LIN {X -0.019,Y -142.969,Z 1935.171,A 0.000,B 0.000,C 90.000,E1 210.846} C_DIS
LIN {X 0.034,Y -141.596,Z 1935.151,A 0.000,B 0.000,C 90.000,E1 207.129} C_DIS
LIN {X -0.051,Y -139.421,Z 1935.115,A 0.000,B 0.000,C 90.000,E1 200.663} C_DIS
LIN {X 0.000,Y -139.148,Z 1935.104,A 0.000,B 0.000,C 90.000,E1 198.779} C_DIS
LIN {X 0.022,Y -138.345,Z 1935.058,A 0.000,B 0.000,C 90.000,E1 190.366} C_DIS
LIN {X 0.008,Y -139.487,Z 1935.006,A 0.000,B 0.000,C 90.000,E1 181.031} C_DIS
LIN {X -0.052,Y -141.088,Z 1934.975,A 0.000,B 0.000,C 90.000,E1 175.469} C_DIS
LIN {X 0.043,Y -142.466,Z 1934.959,A 0.000,B 0.000,C 90.000,E1 172.648} C_DIS
LIN {X -0.009,Y -144.710,Z 1934.934,A 0.000,B 0.000,C 90.000,E1 168.049} C_DIS
LIN {X -0.058,Y -147.309,Z 1934.913,A 0.000,B 0.000,C 90.000,E1 164.393} C_DIS
LIN {X -0.043,Y -150.630,Z 1934.888,A 0.000,B 0.000,C 90.000,E1 159.826} C_DIS
LIN {X 0.033,Y -154.106,Z 1934.868,A 0.000,B 0.000,C 90.000,E1 156.177} C_DIS
LIN {X -0.042,Y -157.530,Z 1934.848,A 0.000,B 0.000,C 90.000,E1 152.615} C_DIS
LIN {X -0.099,Y -161.765,Z 1934.828,A 0.000,B 0.000,C 90.000,E1 149.076} C_DIS
LIN {X 0.007,Y -165.958,Z 1934.808,A 0.000,B 0.000,C 90.000,E1 145.515} C_DIS
LIN {X 0.003,Y -170.951,Z 1934.789,A 0.000,B 0.000,C 90.000,E1 142.029} C_DIS
LIN {X 0.055,Y -175.820,Z 1934.770,A 0.000,B 0.000,C 90.000,E1 138.566} C_DIS
LIN {X 0.051,Y -181.426,Z 1934.751,A 0.000,B 0.000,C 90.000,E1 135.162} C_DIS
LIN {X -0.075,Y -186.930,Z 1934.732,A 0.000,B 0.000,C 90.000,E1 131.838} C_DIS
LIN {X -0.003,Y -191.509,Z 1934.719,A 0.000,B 0.000,C 90.000,E1 129.322} C_DIS
LIN {X 0.082,Y -197.374,Z 1934.700,A 0.000,B 0.000,C 90.000,E1 126.011} C_DIS
LIN {X 0.007,Y -200.649,Z 1934.691,A 0.000,B 0.000,C 90.000,E1 124.405} C_DIS
LIN {X -0.083,Y -206.533,Z 1934.673,A 0.000,B 0.000,C 90.000,E1 121.209} C_DIS
LIN {X 0.011,Y -209.824,Z 1934.664,A 0.000,B 0.000,C 90.000,E1 119.589} C_DIS
LIN {X -0.063,Y -217.182,Z 1934.642,A 0.000,B 0.000,C 90.000,E1 115.668} C_DIS
LIN {X -0.110,Y -218.809,Z 1934.638,A 0.000,B 0.000,C 90.000,E1 114.899} C_DIS
LIN {X 0.031,Y -224.195,Z 1934.621,A 0.000,B 0.000,C 90.000,E1 111.791} C_DIS
LIN {X 0.113,Y -284.154,Z 1934.621,A 0.000,B 0.000,C 90.000,E1 111.770} C_DIS
LIN {X 0.017,Y -285.333,Z 1934.621,A 0.000,B 0.000,C 90.000,E1 111.770} C_DIS
LIN {X -0.012,Y -288.714,Z 1934.620,A 0.000,B 0.000,C 90.000,E1 111.642} C_DIS
LIN {X -0.078,Y -291.984,Z 1934.619,A 0.000,B 0.000,C 90.000,E1 111.408} C_DIS
LIN {X 0.114,Y -295.661,Z 1934.616,A 0.000,B 0.000,C 90.000,E1 110.918} C_DIS
LIN {X -0.073,Y -310.921,Z 1934.602,A 0.000,B 0.000,C 90.000,E1 108.308} C_DIS
LIN {X 0.068,Y -325.651,Z 1934.589,A 0.000,B 0.000,C 90.000,E1 106.024} C_DIS
LIN {X 0.158,Y -339.472,Z 1934.579,A 0.000,B 0.000,C 90.000,E1 104.120} C_DIS
LIN {X 0.015,Y -354.484,Z 1934.568,A 0.000,B 0.000,C 90.000,E1 102.299} C_DIS
LIN {X 0.159,Y -372.954,Z 1934.557,A 0.000,B 0.000,C 90.000,E1 100.254} C_DIS
LIN {X -0.077,Y -391.821,Z 1934.547,A 0.000,B 0.000,C 90.000,E1 98.454} C_DIS
LIN {X -0.060,Y -411.099,Z 1934.538,A 0.000,B 0.000,C 90.000,E1 96.777} C_DIS
LIN {X -0.118,Y -433.506,Z 1934.528,A 0.000,B 0.000,C 90.000,E1 95.049} C_DIS
LIN {X -0.139,Y -439.166,Z 1934.526,A 0.000,B 0.000,C 90.000,E1 94.645} C_DIS
LIN {X -0.149,Y -443.334,Z 1934.523,A 0.000,B 0.000,C 90.000,E1 94.245} C_DIS
LIN {X 0.181,Y -445.054,Z 1934.522,A 0.000,B 0.000,C 90.000,E1 93.955} C_DIS
LIN {X 0.036,Y -446.375,Z 1934.521,A 0.000,B 0.000,C 90.000,E1 93.726} C_DIS
LIN {X -0.039,Y -448.200,Z 1934.518,A 0.000,B 0.000,C 90.000,E1 93.212} C_DIS
LIN {X -0.081,Y -448.963,Z 1934.515,A 0.000,B 0.000,C 90.000,E1 92.694} C_DIS
LIN {X -0.135,Y -448.790,Z 1934.512,A 0.000,B 0.000,C 90.000,E1 92.178} C_DIS
LIN {X -0.168,Y -447.662,Z 1934.509,A 0.000,B 0.000,C 90.000,E1 91.661} C_DIS
LIN {X 0.032,Y -446.690,Z 1934.508,A 0.000,B 0.000,C 90.000,E1 91.375} C_DIS
LIN {X -0.216,Y -445.387,Z 1934.506,A 0.000,B 0.000,C 90.000,E1 91.146} C_DIS
LIN {X 0.160,Y -433.910,Z 1934.496,A 0.000,B 0.000,C 90.000,E1 89.255} C_DIS
LIN {X 0.177,Y -423.887,Z 1934.487,A 0.000,B 0.000,C 90.000,E1 87.650} C_DIS
LIN {X 0.137,Y -412.109,Z 1934.477,A 0.000,B 0.000,C 90.000,E1 85.755} C_DIS
LIN {X -0.196,Y -401.950,Z 1934.467,A 0.000,B 0.000,C 90.000,E1 84.147} C_DIS
LIN {X -0.211,Y -389.964,Z 1934.456,A 0.000,B 0.000,C 90.000,E1 82.186} C_DIS
LIN {X 0.022,Y -378.082,Z 1934.445,A 0.000,B 0.000,C 90.000,E1 80.151} C_DIS
LIN {X 0.037,Y -363.093,Z 1934.431,A 0.000,B 0.000,C 90.000,E1 77.521} C_DIS
LIN {X 0.108,Y -345.897,Z 1934.412,A 0.000,B 0.000,C 90.000,E1 74.212} C_DIS
LIN {X 0.052,Y -333.963,Z 1934.399,A 0.000,B 0.000,C 90.000,E1 71.764} C_DIS
LIN {X 0.061,Y -323.718,Z 1934.387,A 0.000,B 0.000,C 90.000,E1 69.571} C_DIS
LIN {X 0.153,Y -309.663,Z 1934.369,A 0.000,B 0.000,C 90.000,E1 66.357} C_DIS
LIN {X 0.003,Y -300.191,Z 1934.356,A 0.000,B 0.000,C 90.000,E1 64.101} C_DIS
LIN {X -0.115,Y -288.155,Z 1934.339,A 0.000,B 0.000,C 90.000,E1 61.129} C_DIS
LIN {X -0.015,Y -280.090,Z 1934.328,A 0.000,B 0.000,C 90.000,E1 59.076} C_DIS
LIN {X 0.158,Y -270.556,Z 1934.315,A 0.000,B 0.000,C 90.000,E1 56.628} C_DIS
LIN {X 0.074,Y -263.707,Z 1934.305,A 0.000,B 0.000,C 90.000,E1 54.895} C_DIS
LIN {X -0.006,Y -252.710,Z 1934.289,A 0.000,B 0.000,C 90.000,E1 52.065} C_DIS
LIN {X -0.086,Y -243.127,Z 1934.275,A 0.000,B 0.000,C 90.000,E1 49.542} C_DIS
LIN {X 0.066,Y -232.480,Z 1934.259,A 0.000,B 0.000,C 90.000,E1 46.539} C_DIS
LIN {X -0.064,Y -222.206,Z 1934.242,A 0.000,B 0.000,C 90.000,E1 43.542} C_DIS
LIN {X 0.099,Y -211.300,Z 1934.222,A 0.000,B 0.000,C 90.000,E1 40.011} C_DIS
LIN {X -0.042,Y -203.498,Z 1934.207,A 0.000,B 0.000,C 90.000,E1 37.282} C_DIS
LIN {X -0.047,Y -195.382,Z 1934.189,A 0.000,B 0.000,C 90.000,E1 34.072} C_DIS
LIN {X -0.029,Y -188.013,Z 1934.171,A 0.000,B 0.000,C 90.000,E1 30.797} C_DIS
LIN {X 0.006,Y -181.382,Z 1934.153,A 0.000,B 0.000,C 90.000,E1 27.462} C_DIS
LIN {X -0.041,Y -176.866,Z 1934.139,A 0.000,B 0.000,C 90.000,E1 24.951} C_DIS
LIN {X -0.019,Y -171.587,Z 1934.120,A 0.000,B 0.000,C 90.000,E1 21.535} C_DIS
LIN {X 0.071,Y -167.096,Z 1934.100,A 0.000,B 0.000,C 90.000,E1 18.055} C_DIS
LIN {X 0.002,Y -163.458,Z 1934.081,A 0.000,B 0.000,C 90.000,E1 14.592} C_DIS
LIN {X -0.011,Y -159.746,Z 1934.057,A 0.000,B 0.000,C 90.000,E1 10.197} C_DIS
LIN {X 0.050,Y -157.186,Z 1934.032,A 0.000,B 0.000,C 90.000,E1 5.739} C_DIS
LIN {X -0.028,Y -154.901,Z 1933.997,A 0.000,B 0.000,C 90.000,E1 359.542} C_DIS
LIN {X 0.057,Y -154.146,Z 1933.953,A 0.000,B 0.000,C 90.000,E1 351.432} C_DIS
LIN {X -0.021,Y -155.869,Z 1933.913,A 0.000,B 0.000,C 90.000,E1 344.283} C_DIS
LIN {X 0.041,Y -158.583,Z 1933.883,A 0.000,B 0.000,C 90.000,E1 338.901} C_DIS
LIN {X 0.055,Y -162.176,Z 1933.858,A 0.000,B 0.000,C 90.000,E1 334.460} C_DIS
LIN {X -0.038,Y -166.049,Z 1933.839,A 0.000,B 0.000,C 90.000,E1 330.973} C_DIS
LIN {X 0.060,Y -170.918,Z 1933.819,A 0.000,B 0.000,C 90.000,E1 327.454} C_DIS
LIN {X -0.028,Y -175.211,Z 1933.805,A 0.000,B 0.000,C 90.000,E1 324.895} C_DIS
LIN {X 0.023,Y -180.173,Z 1933.791,A 0.000,B 0.000,C 90.000,E1 322.316} C_DIS
LIN {X 0.022,Y -186.029,Z 1933.777,A 0.000,B 0.000,C 90.000,E1 319.784} C_DIS
LIN {X -0.012,Y -191.640,Z 1933.765,A 0.000,B 0.000,C 90.000,E1 317.715} C_DIS
LIN {X 0.024,Y -199.313,Z 1933.751,A 0.000,B 0.000,C 90.000,E1 315.243} C_DIS
LIN {X -0.075,Y -207.901,Z 1933.738,A 0.000,B 0.000,C 90.000,E1 312.852} C_DIS
LIN {X -0.095,Y -218.960,Z 1933.723,A 0.000,B 0.000,C 90.000,E1 310.092} C_DIS
LIN {X -0.031,Y -232.882,Z 1933.705,A 0.000,B 0.000,C 90.000,E1 306.996} C_DIS
LIN {X 0.030,Y -247.942,Z 1933.689,A 0.000,B 0.000,C 90.000,E1 303.992} C_DIS
LIN {X 0.080,Y -259.865,Z 1933.677,A 0.000,B 0.000,C 90.000,E1 301.799} C_DIS
LIN {X 0.084,Y -271.928,Z 1933.665,A 0.000,B 0.000,C 90.000,E1 299.667} C_DIS
LIN {X -0.143,Y -281.824,Z 1933.655,A 0.000,B 0.000,C 90.000,E1 297.975} C_DIS
LIN {X 0.029,Y -291.425,Z 1933.646,A 0.000,B 0.000,C 90.000,E1 296.232} C_DIS
LIN {X 0.109,Y -296.837,Z 1933.640,A 0.000,B 0.000,C 90.000,E1 295.207} C_DIS
LIN {X 0.110,Y -301.639,Z 1933.635,A 0.000,B 0.000,C 90.000,E1 294.207} C_DIS
LIN {X -0.004,Y -304.447,Z 1933.631,A 0.000,B 0.000,C 90.000,E1 293.567} C_DIS
LIN {X 0.057,Y -306.850,Z 1933.627,A 0.000,B 0.000,C 90.000,E1 292.898} C_DIS
LIN {X -0.030,Y -308.861,Z 1933.624,A 0.000,B 0.000,C 90.000,E1 292.259} C_DIS
LIN {X 0.058,Y -310.530,Z 1933.620,A 0.000,B 0.000,C 90.000,E1 291.589} C_DIS
LIN {X -0.129,Y -311.874,Z 1933.616,A 0.000,B 0.000,C 90.000,E1 290.972} C_DIS
LIN {X -0.014,Y -312.871,Z 1933.613,A 0.000,B 0.000,C 90.000,E1 290.301} C_DIS
LIN {X 0.111,Y -313.512,Z 1933.609,A 0.000,B 0.000,C 90.000,E1 289.631} C_DIS
LIN {X -0.158,Y -313.857,Z 1933.606,A 0.000,B 0.000,C 90.000,E1 289.033} C_DIS
LIN {X -0.023,Y -313.847,Z 1933.602,A 0.000,B 0.000,C 90.000,E1 288.362} C_DIS
LIN {X 0.111,Y -313.460,Z 1933.598,A 0.000,B 0.000,C 90.000,E1 287.692} C_DIS
LIN {X 0.150,Y -312.644,Z 1933.595,A 0.000,B 0.000,C 90.000,E1 287.040} C_DIS
LIN {X -0.110,Y -311.343,Z 1933.591,A 0.000,B 0.000,C 90.000,E1 286.441} C_DIS
LIN {X -0.075,Y -309.501,Z 1933.588,A 0.000,B 0.000,C 90.000,E1 285.788} C_DIS
LIN {X -0.048,Y -307.046,Z 1933.584,A 0.000,B 0.000,C 90.000,E1 285.134} C_DIS
LIN {X -0.039,Y -303.810,Z 1933.580,A 0.000,B 0.000,C 90.000,E1 284.481} C_DIS
LIN {X -0.081,Y -296.077,Z 1933.573,A 0.000,B 0.000,C 90.000,E1 283.175} C_DIS
LIN {X 0.005,Y -290.833,Z 1933.568,A 0.000,B 0.000,C 90.000,E1 282.187} C_DIS
LIN {X -0.087,Y -286.473,Z 1933.564,A 0.000,B 0.000,C 90.000,E1 281.535} C_DIS
LIN {X 0.018,Y -281.136,Z 1933.560,A 0.000,B 0.000,C 90.000,E1 280.838} C_DIS
LIN {X 0.016,Y -274.907,Z 1933.557,A 0.000,B 0.000,C 90.000,E1 280.197} C_DIS
LIN {X 0.068,Y -268.464,Z 1933.553,A 0.000,B 0.000,C 90.000,E1 279.613} C_DIS
LIN {X -0.143,Y -261.822,Z 1933.551,A 0.000,B 0.000,C 90.000,E1 279.151} C_DIS
LIN {X -0.032,Y -255.092,Z 1933.548,A 0.000,B 0.000,C 90.000,E1 278.681} C_DIS
LIN {X 0.029,Y -248.149,Z 1933.546,A 0.000,B 0.000,C 90.000,E1 278.276} C_DIS
LIN {X 0.084,Y -240.671,Z 1933.544,A 0.000,B 0.000,C 90.000,E1 277.936} C_DIS
LIN {X -0.018,Y -232.620,Z 1933.543,A 0.000,B 0.000,C 90.000,E1 277.701} C_DIS
LIN {X -0.096,Y -221.950,Z 1933.542,A 0.000,B 0.000,C 90.000,E1 277.530} C_DIS
LIN {X -0.033,Y -216.160,Z 1933.541,A 0.000,B 0.000,C 90.000,E1 277.466} C_DIS
LIN {X -0.058,Y -180.199,Z 1933.541,A 0.000,B 0.000,C 90.000,E1 277.466} C_DIS
LIN {X 0.058,Y -181.027,Z 1933.530,A 0.000,B 0.000,C 90.000,E1 275.391} C_DIS
LIN {X 0.033,Y -181.578,Z 1933.502,A 0.000,B 0.000,C 90.000,E1 270.344} C_DIS
LIN {X 0.009,Y -180.904,Z 1933.474,A 0.000,B 0.000,C 90.000,E1 265.298} C_DIS
LIN {X -0.042,Y -180.245,Z 1933.464,A 0.000,B 0.000,C 90.000,E1 263.628} C_DIS
LIN {X -0.023,Y -178.732,Z 1933.441,A 0.000,B 0.000,C 90.000,E1 259.398} C_DIS
LIN {X 0.045,Y -175.780,Z 1933.413,A 0.000,B 0.000,C 90.000,E1 254.283} C_DIS
LIN {X 0.032,Y -171.964,Z 1933.384,A 0.000,B 0.000,C 90.000,E1 249.156} C_DIS
LIN {X 0.069,Y -171.361,Z 1933.380,A 0.000,B 0.000,C 90.000,E1 248.284} C_DIS
LIN {X 0.046,Y -167.610,Z 1933.355,A 0.000,B 0.000,C 90.000,E1 243.973} C_DIS
LIN {X 0.059,Y -166.257,Z 1933.346,A 0.000,B 0.000,C 90.000,E1 242.231} C_DIS
LIN {X 0.046,Y -163.011,Z 1933.326,A 0.000,B 0.000,C 90.000,E1 238.742} C_DIS
LIN {X -0.040,Y -160.934,Z 1933.312,A 0.000,B 0.000,C 90.000,E1 236.135} C_DIS
LIN {X 0.069,Y -157.694,Z 1933.292,A 0.000,B 0.000,C 90.000,E1 232.557} C_DIS
LIN {X 0.008,Y -155.733,Z 1933.277,A 0.000,B 0.000,C 90.000,E1 229.908} C_DIS
LIN {X 0.061,Y -151.992,Z 1933.252,A 0.000,B 0.000,C 90.000,E1 225.405} C_DIS
LIN {X 0.077,Y -150.237,Z 1933.237,A 0.000,B 0.000,C 90.000,E1 222.690} C_DIS
LIN {X -0.001,Y -146.997,Z 1933.212,A 0.000,B 0.000,C 90.000,E1 218.177} C_DIS
LIN {X -0.010,Y -145.582,Z 1933.197,A 0.000,B 0.000,C 90.000,E1 215.438} C_DIS
LIN {X -0.016,Y -142.970,Z 1933.171,A 0.000,B 0.000,C 90.000,E1 210.846} C_DIS
LIN {X 0.037,Y -141.597,Z 1933.151,A 0.000,B 0.000,C 90.000,E1 207.129} C_DIS
LIN {X -0.046,Y -139.422,Z 1933.115,A 0.000,B 0.000,C 90.000,E1 200.663} C_DIS
LIN {X 0.004,Y -139.150,Z 1933.104,A 0.000,B 0.000,C 90.000,E1 198.779} C_DIS
LIN {X 0.026,Y -138.346,Z 1933.058,A 0.000,B 0.000,C 90.000,E1 190.366} C_DIS
LIN {X 0.012,Y -139.487,Z 1933.006,A 0.000,B 0.000,C 90.000,E1 181.031} C_DIS
LIN {X -0.048,Y -141.088,Z 1932.975,A 0.000,B 0.000,C 90.000,E1 175.469} C_DIS
LIN {X 0.047,Y -142.464,Z 1932.959,A 0.000,B 0.000,C 90.000,E1 172.648} C_DIS
LIN {X -0.005,Y -144.709,Z 1932.934,A 0.000,B 0.000,C 90.000,E1 168.049} C_DIS
LIN {X -0.054,Y -147.308,Z 1932.913,A 0.000,B 0.000,C 90.000,E1 164.393} C_DIS
LIN {X -0.039,Y -150.628,Z 1932.888,A 0.000,B 0.000,C 90.000,E1 159.826} C_DIS
LIN {X 0.037,Y -154.105,Z 1932.868,A 0.000,B 0.000,C 90.000,E1 156.177} C_DIS
LIN {X -0.039,Y -157.528,Z 1932.848,A 0.000,B 0.000,C 90.000,E1 152.615} C_DIS
LIN {X -0.095,Y -161.763,Z 1932.828,A 0.000,B 0.000,C 90.000,E1 149.076} C_DIS
LIN {X 0.011,Y -165.957,Z 1932.808,A 0.000,B 0.000,C 90.000,E1 145.515} C_DIS
LIN {X 0.008,Y -170.948,Z 1932.789,A 0.000,B 0.000,C 90.000,E1 142.029} C_DIS
LIN {X 0.059,Y -175.817,Z 1932.770,A 0.000,B 0.000,C 90.000,E1 138.566} C_DIS
LIN {X 0.055,Y -181.424,Z 1932.751,A 0.000,B 0.000,C 90.000,E1 135.162} C_DIS
LIN {X -0.071,Y -186.929,Z 1932.732,A 0.000,B 0.000,C 90.000,E1 131.838} C_DIS
LIN {X 0.002,Y -191.506,Z 1932.719,A 0.000,B 0.000,C 90.000,E1 129.322} C_DIS
LIN {X 0.087,Y -197.371,Z 1932.700,A 0.000,B 0.000,C 90.000,E1 126.011} C_DIS
LIN {X 0.011,Y -200.647,Z 1932.691,A 0.000,B 0.000,C 90.000,E1 124.405} C_DIS
LIN {X -0.079,Y -206.530,Z 1932.673,A 0.000,B 0.000,C 90.000,E1 121.209} C_DIS
LIN {X 0.015,Y -209.822,Z 1932.664,A 0.000,B 0.000,C 90.000,E1 119.589} C_DIS
LIN {X -0.059,Y -217.180,Z 1932.642,A 0.000,B 0.000,C 90.000,E1 115.668} C_DIS
LIN {X -0.105,Y -218.806,Z 1932.638,A 0.000,B 0.000,C 90.000,E1 114.899} C_DIS
LIN {X 0.036,Y -224.194,Z 1932.621,A 0.000,B 0.000,C 90.000,E1 111.791} C_DIS
LIN {X 0.119,Y -284.134,Z 1932.621,A 0.000,B 0.000,C 90.000,E1 111.770} C_DIS
LIN {X 0.022,Y -285.319,Z 1932.621,A 0.000,B 0.000,C 90.000,E1 111.770} C_DIS
LIN {X -0.003,Y -288.698,Z 1932.620,A 0.000,B 0.000,C 90.000,E1 111.642} C_DIS
LIN {X -0.068,Y -291.966,Z 1932.619,A 0.000,B 0.000,C 90.000,E1 111.408} C_DIS
LIN {X 0.128,Y -295.643,Z 1932.616,A 0.000,B 0.000,C 90.000,E1 110.918} C_DIS
LIN {X -0.056,Y -310.901,Z 1932.602,A 0.000,B 0.000,C 90.000,E1 108.308} C_DIS
LIN {X 0.087,Y -325.627,Z 1932.589,A 0.000,B 0.000,C 90.000,E1 106.024} C_DIS
LIN {X 0.176,Y -339.447,Z 1932.579,A 0.000,B 0.000,C 90.000,E1 104.120} C_DIS
LIN {X 0.035,Y -354.456,Z 1932.568,A 0.000,B 0.000,C 90.000,E1 102.299} C_DIS
LIN {X 0.176,Y -372.924,Z 1932.557,A 0.000,B 0.000,C 90.000,E1 100.254} C_DIS
LIN {X -0.060,Y -391.792,Z 1932.547,A 0.000,B 0.000,C 90.000,E1 98.454} C_DIS
LIN {X -0.043,Y -411.070,Z 1932.538,A 0.000,B 0.000,C 90.000,E1 96.777} C_DIS
LIN {X -0.102,Y -433.476,Z 1932.528,A 0.000,B 0.000,C 90.000,E1 95.049} C_DIS
LIN {X -0.123,Y -439.135,Z 1932.526,A 0.000,B 0.000,C 90.000,E1 94.645} C_DIS
LIN {X -0.134,Y -443.311,Z 1932.523,A 0.000,B 0.000,C 90.000,E1 94.245} C_DIS
LIN {X 0.198,Y -445.032,Z 1932.522,A 0.000,B 0.000,C 90.000,E1 93.955} C_DIS
LIN {X 0.055,Y -446.353,Z 1932.521,A 0.000,B 0.000,C 90.000,E1 93.726} C_DIS
LIN {X -0.020,Y -448.182,Z 1932.518,A 0.000,B 0.000,C 90.000,E1 93.212} C_DIS
LIN {X -0.062,Y -448.948,Z 1932.515,A 0.000,B 0.000,C 90.000,E1 92.694} C_DIS
LIN {X -0.116,Y -448.778,Z 1932.512,A 0.000,B 0.000,C 90.000,E1 92.178} C_DIS
LIN {X -0.149,Y -447.653,Z 1932.509,A 0.000,B 0.000,C 90.000,E1 91.661} C_DIS
LIN {X 0.050,Y -446.682,Z 1932.508,A 0.000,B 0.000,C 90.000,E1 91.375} C_DIS
LIN {X -0.197,Y -445.381,Z 1932.506,A 0.000,B 0.000,C 90.000,E1 91.146} C_DIS
LIN {X 0.178,Y -433.905,Z 1932.496,A 0.000,B 0.000,C 90.000,E1 89.255} C_DIS
LIN {X 0.194,Y -423.883,Z 1932.487,A 0.000,B 0.000,C 90.000,E1 87.650} C_DIS
LIN {X 0.154,Y -412.105,Z 1932.477,A 0.000,B 0.000,C 90.000,E1 85.755} C_DIS
LIN {X -0.180,Y -401.947,Z 1932.467,A 0.000,B 0.000,C 90.000,E1 84.147} C_DIS
LIN {X -0.195,Y -389.961,Z 1932.456,A 0.000,B 0.000,C 90.000,E1 82.186} C_DIS
LIN {X 0.037,Y -378.076,Z 1932.445,A 0.000,B 0.000,C 90.000,E1 80.151} C_DIS
LIN {X 0.052,Y -363.086,Z 1932.431,A 0.000,B 0.000,C 90.000,E1 77.521} C_DIS
LIN {X 0.122,Y -345.888,Z 1932.412,A 0.000,B 0.000,C 90.000,E1 74.212} C_DIS
LIN {X 0.065,Y -333.955,Z 1932.399,A 0.000,B 0.000,C 90.000,E1 71.764} C_DIS
LIN {X 0.074,Y -323.708,Z 1932.387,A 0.000,B 0.000,C 90.000,E1 69.571} C_DIS
LIN {X 0.165,Y -309.651,Z 1932.369,A 0.000,B 0.000,C 90.000,E1 66.357} C_DIS
LIN {X 0.015,Y -300.178,Z 1932.356,A 0.000,B 0.000,C 90.000,E1 64.101} C_DIS
LIN {X -0.105,Y -288.140,Z 1932.339,A 0.000,B 0.000,C 90.000,E1 61.129} C_DIS
LIN {X -0.005,Y -280.075,Z 1932.328,A 0.000,B 0.000,C 90.000,E1 59.076} C_DIS
LIN {X 0.167,Y -270.544,Z 1932.315,A 0.000,B 0.000,C 90.000,E1 56.628} C_DIS
LIN {X 0.082,Y -263.695,Z 1932.305,A 0.000,B 0.000,C 90.000,E1 54.895} C_DIS
LIN {X 0.002,Y -252.701,Z 1932.289,A 0.000,B 0.000,C 90.000,E1 52.065} C_DIS
LIN {X -0.079,Y -243.117,Z 1932.275,A 0.000,B 0.000,C 90.000,E1 49.542} C_DIS
LIN {X 0.072,Y -232.468,Z 1932.259,A 0.000,B 0.000,C 90.000,E1 46.539} C_DIS
LIN {X -0.058,Y -222.193,Z 1932.242,A 0.000,B 0.000,C 90.000,E1 43.542} C_DIS
LIN {X 0.104,Y -211.288,Z 1932.222,A 0.000,B 0.000,C 90.000,E1 40.011} C_DIS
LIN {X -0.037,Y -203.488,Z 1932.207,A 0.000,B 0.000,C 90.000,E1 37.282} C_DIS
LIN {X -0.042,Y -195.374,Z 1932.189,A 0.000,B 0.000,C 90.000,E1 34.072} C_DIS
LIN {X -0.024,Y -188.008,Z 1932.171,A 0.000,B 0.000,C 90.000,E1 30.797} C_DIS
LIN {X 0.010,Y -181.376,Z 1932.153,A 0.000,B 0.000,C 90.000,E1 27.462} C_DIS
LIN {X -0.037,Y -176.860,Z 1932.139,A 0.000,B 0.000,C 90.000,E1 24.951} C_DIS
LIN {X -0.015,Y -171.583,Z 1932.120,A 0.000,B 0.000,C 90.000,E1 21.535} C_DIS
LIN {X 0.074,Y -167.091,Z 1932.100,A 0.000,B 0.000,C 90.000,E1 18.055} C_DIS
LIN {X 0.005,Y -163.452,Z 1932.081,A 0.000,B 0.000,C 90.000,E1 14.592} C_DIS
LIN {X -0.008,Y -159.739,Z 1932.057,A 0.000,B 0.000,C 90.000,E1 10.197} C_DIS
LIN {X 0.052,Y -157.177,Z 1932.032,A 0.000,B 0.000,C 90.000,E1 5.739} C_DIS
LIN {X -0.028,Y -154.892,Z 1931.997,A 0.000,B 0.000,C 90.000,E1 359.542} C_DIS
LIN {X -0.004,Y -154.217,Z 1931.948,A 0.000,B 0.000,C 90.000,E1 350.557} C_DIS
LIN {X 0.005,Y -156.202,Z 1931.908,A 0.000,B 0.000,C 90.000,E1 343.378} C_DIS
LIN {X 0.040,Y -158.579,Z 1931.883,A 0.000,B 0.000,C 90.000,E1 338.901} C_DIS
LIN {X 0.055,Y -162.174,Z 1931.858,A 0.000,B 0.000,C 90.000,E1 334.460} C_DIS
LIN {X -0.039,Y -166.051,Z 1931.839,A 0.000,B 0.000,C 90.000,E1 330.973} C_DIS
LIN {X 0.059,Y -170.923,Z 1931.819,A 0.000,B 0.000,C 90.000,E1 327.454} C_DIS
LIN {X -0.030,Y -175.218,Z 1931.805,A 0.000,B 0.000,C 90.000,E1 324.895} C_DIS
LIN {X 0.023,Y -180.180,Z 1931.791,A 0.000,B 0.000,C 90.000,E1 322.316} C_DIS
LIN {X 0.021,Y -186.038,Z 1931.777,A 0.000,B 0.000,C 90.000,E1 319.784} C_DIS
LIN {X -0.014,Y -191.649,Z 1931.765,A 0.000,B 0.000,C 90.000,E1 317.715} C_DIS
LIN {X 0.024,Y -199.318,Z 1931.751,A 0.000,B 0.000,C 90.000,E1 315.243} C_DIS
LIN {X -0.075,Y -207.907,Z 1931.738,A 0.000,B 0.000,C 90.000,E1 312.852} C_DIS
LIN {X -0.095,Y -218.968,Z 1931.723,A 0.000,B 0.000,C 90.000,E1 310.092} C_DIS
LIN {X -0.031,Y -232.892,Z 1931.705,A 0.000,B 0.000,C 90.000,E1 306.996} C_DIS
LIN {X 0.031,Y -247.952,Z 1931.689,A 0.000,B 0.000,C 90.000,E1 303.992} C_DIS
LIN {X 0.080,Y -259.876,Z 1931.677,A 0.000,B 0.000,C 90.000,E1 301.799} C_DIS
LIN {X 0.085,Y -271.939,Z 1931.665,A 0.000,B 0.000,C 90.000,E1 299.667} C_DIS
LIN {X -0.142,Y -281.832,Z 1931.655,A 0.000,B 0.000,C 90.000,E1 297.975} C_DIS
LIN {X 0.030,Y -291.433,Z 1931.646,A 0.000,B 0.000,C 90.000,E1 296.232} C_DIS
LIN {X 0.110,Y -296.850,Z 1931.640,A 0.000,B 0.000,C 90.000,E1 295.207} C_DIS
LIN {X 0.112,Y -301.653,Z 1931.635,A 0.000,B 0.000,C 90.000,E1 294.207} C_DIS
LIN {X -0.004,Y -304.459,Z 1931.631,A 0.000,B 0.000,C 90.000,E1 293.567} C_DIS
LIN {X 0.058,Y -306.863,Z 1931.627,A 0.000,B 0.000,C 90.000,E1 292.898} C_DIS
LIN {X -0.029,Y -308.873,Z 1931.624,A 0.000,B 0.000,C 90.000,E1 292.259} C_DIS
LIN {X 0.060,Y -310.545,Z 1931.620,A 0.000,B 0.000,C 90.000,E1 291.589} C_DIS
LIN {X -0.127,Y -311.888,Z 1931.616,A 0.000,B 0.000,C 90.000,E1 290.972} C_DIS
LIN {X -0.012,Y -312.887,Z 1931.613,A 0.000,B 0.000,C 90.000,E1 290.301} C_DIS
LIN {X 0.112,Y -313.527,Z 1931.609,A 0.000,B 0.000,C 90.000,E1 289.631} C_DIS
LIN {X -0.156,Y -313.871,Z 1931.606,A 0.000,B 0.000,C 90.000,E1 289.033} C_DIS
LIN {X -0.021,Y -313.861,Z 1931.602,A 0.000,B 0.000,C 90.000,E1 288.362} C_DIS
LIN {X 0.114,Y -313.474,Z 1931.598,A 0.000,B 0.000,C 90.000,E1 287.692} C_DIS
LIN {X 0.152,Y -312.661,Z 1931.595,A 0.000,B 0.000,C 90.000,E1 287.040} C_DIS
LIN {X -0.108,Y -311.362,Z 1931.591,A 0.000,B 0.000,C 90.000,E1 286.441} C_DIS
LIN {X -0.073,Y -309.518,Z 1931.588,A 0.000,B 0.000,C 90.000,E1 285.788} C_DIS
LIN {X -0.046,Y -307.064,Z 1931.584,A 0.000,B 0.000,C 90.000,E1 285.134} C_DIS
LIN {X -0.036,Y -303.828,Z 1931.580,A 0.000,B 0.000,C 90.000,E1 284.481} C_DIS
LIN {X -0.079,Y -296.098,Z 1931.573,A 0.000,B 0.000,C 90.000,E1 283.175} C_DIS
LIN {X 0.009,Y -290.846,Z 1931.568,A 0.000,B 0.000,C 90.000,E1 282.187} C_DIS
LIN {X -0.082,Y -286.490,Z 1931.564,A 0.000,B 0.000,C 90.000,E1 281.535} C_DIS
LIN {X 0.023,Y -281.149,Z 1931.560,A 0.000,B 0.000,C 90.000,E1 280.838} C_DIS
LIN {X 0.020,Y -274.914,Z 1931.557,A 0.000,B 0.000,C 90.000,E1 280.197} C_DIS
LIN {X 0.072,Y -268.472,Z 1931.553,A 0.000,B 0.000,C 90.000,E1 279.613} C_DIS
LIN {X -0.140,Y -261.831,Z 1931.551,A 0.000,B 0.000,C 90.000,E1 279.151} C_DIS
LIN {X -0.027,Y -255.106,Z 1931.548,A 0.000,B 0.000,C 90.000,E1 278.681} C_DIS
LIN {X 0.034,Y -248.163,Z 1931.546,A 0.000,B 0.000,C 90.000,E1 278.276} C_DIS
LIN {X 0.089,Y -240.685,Z 1931.544,A 0.000,B 0.000,C 90.000,E1 277.936} C_DIS
LIN {X -0.012,Y -232.646,Z 1931.543,A 0.000,B 0.000,C 90.000,E1 277.701} C_DIS
LIN {X -0.092,Y -221.965,Z 1931.542,A 0.000,B 0.000,C 90.000,E1 277.530} C_DIS
LIN {X -0.028,Y -216.198,Z 1931.541,A 0.000,B 0.000,C 90.000,E1 277.466} C_DIS
LIN {X -0.054,Y -180.199,Z 1931.541,A 0.000,B 0.000,C 90.000,E1 277.466} C_DIS
LIN {X 0.062,Y -181.028,Z 1931.530,A 0.000,B 0.000,C 90.000,E1 275.391} C_DIS
LIN {X 0.037,Y -181.578,Z 1931.502,A 0.000,B 0.000,C 90.000,E1 270.344} C_DIS
LIN {X 0.013,Y -180.904,Z 1931.474,A 0.000,B 0.000,C 90.000,E1 265.298} C_DIS
LIN {X -0.038,Y -180.246,Z 1931.464,A 0.000,B 0.000,C 90.000,E1 263.628} C_DIS
LIN {X -0.019,Y -178.734,Z 1931.441,A 0.000,B 0.000,C 90.000,E1 259.398} C_DIS
LIN {X 0.049,Y -175.781,Z 1931.413,A 0.000,B 0.000,C 90.000,E1 254.283} C_DIS
LIN {X 0.037,Y -171.965,Z 1931.384,A 0.000,B 0.000,C 90.000,E1 249.156} C_DIS
LIN {X 0.073,Y -171.362,Z 1931.380,A 0.000,B 0.000,C 90.000,E1 248.284} C_DIS
LIN {X 0.051,Y -167.611,Z 1931.355,A 0.000,B 0.000,C 90.000,E1 243.973} C_DIS
LIN {X 0.063,Y -166.258,Z 1931.346,A 0.000,B 0.000,C 90.000,E1 242.231} C_DIS
LIN {X 0.050,Y -163.013,Z 1931.326,A 0.000,B 0.000,C 90.000,E1 238.742} C_DIS
LIN {X -0.037,Y -160.936,Z 1931.312,A 0.000,B 0.000,C 90.000,E1 236.135} C_DIS
LIN {X 0.074,Y -157.695,Z 1931.292,A 0.000,B 0.000,C 90.000,E1 232.557} C_DIS
LIN {X 0.011,Y -155.734,Z 1931.277,A 0.000,B 0.000,C 90.000,E1 229.908} C_DIS
LIN {X 0.065,Y -151.993,Z 1931.252,A 0.000,B 0.000,C 90.000,E1 225.405} C_DIS
LIN {X 0.081,Y -150.238,Z 1931.237,A 0.000,B 0.000,C 90.000,E1 222.690} C_DIS
LIN {X 0.004,Y -146.998,Z 1931.212,A 0.000,B 0.000,C 90.000,E1 218.177} C_DIS
LIN {X -0.006,Y -145.582,Z 1931.197,A 0.000,B 0.000,C 90.000,E1 215.438} C_DIS
LIN {X -0.012,Y -142.971,Z 1931.171,A 0.000,B 0.000,C 90.000,E1 210.846} C_DIS
LIN {X 0.041,Y -141.598,Z 1931.151,A 0.000,B 0.000,C 90.000,E1 207.129} C_DIS
LIN {X -0.043,Y -139.422,Z 1931.115,A 0.000,B 0.000,C 90.000,E1 200.663} C_DIS
LIN {X 0.007,Y -139.150,Z 1931.104,A 0.000,B 0.000,C 90.000,E1 198.779} C_DIS
LIN {X 0.029,Y -138.345,Z 1931.058,A 0.000,B 0.000,C 90.000,E1 190.366} C_DIS
LIN {X 0.016,Y -139.486,Z 1931.006,A 0.000,B 0.000,C 90.000,E1 181.031} C_DIS
LIN {X -0.045,Y -141.086,Z 1930.975,A 0.000,B 0.000,C 90.000,E1 175.469} C_DIS
LIN {X 0.051,Y -142.464,Z 1930.959,A 0.000,B 0.000,C 90.000,E1 172.648} C_DIS
LIN {X -0.001,Y -144.709,Z 1930.934,A 0.000,B 0.000,C 90.000,E1 168.049} C_DIS
LIN {X -0.050,Y -147.307,Z 1930.913,A 0.000,B 0.000,C 90.000,E1 164.393} C_DIS
LIN {X -0.035,Y -150.627,Z 1930.888,A 0.000,B 0.000,C 90.000,E1 159.826} C_DIS
LIN {X 0.041,Y -154.103,Z 1930.868,A 0.000,B 0.000,C 90.000,E1 156.177} C_DIS
LIN {X -0.035,Y -157.526,Z 1930.848,A 0.000,B 0.000,C 90.000,E1 152.615} C_DIS
LIN {X -0.090,Y -161.762,Z 1930.828,A 0.000,B 0.000,C 90.000,E1 149.076} C_DIS
LIN {X 0.015,Y -165.954,Z 1930.808,A 0.000,B 0.000,C 90.000,E1 145.515} C_DIS
LIN {X 0.012,Y -170.946,Z 1930.789,A 0.000,B 0.000,C 90.000,E1 142.029} C_DIS
LIN {X -0.069,Y -175.815,Z 1930.770,A 0.000,B 0.000,C 90.000,E1 138.609} C_DIS
LIN {X 0.060,Y -181.422,Z 1930.751,A 0.000,B 0.000,C 90.000,E1 135.162} C_DIS
LIN {X -0.067,Y -186.926,Z 1930.732,A 0.000,B 0.000,C 90.000,E1 131.838} C_DIS
LIN {X 0.006,Y -191.504,Z 1930.719,A 0.000,B 0.000,C 90.000,E1 129.322} C_DIS
LIN {X 0.091,Y -197.368,Z 1930.700,A 0.000,B 0.000,C 90.000,E1 126.011} C_DIS
LIN {X 0.015,Y -200.644,Z 1930.691,A 0.000,B 0.000,C 90.000,E1 124.405} C_DIS
LIN {X -0.074,Y -206.528,Z 1930.673,A 0.000,B 0.000,C 90.000,E1 121.209} C_DIS
LIN {X 0.020,Y -209.819,Z 1930.664,A 0.000,B 0.000,C 90.000,E1 119.589} C_DIS
LIN {X -0.054,Y -217.177,Z 1930.643,A 0.000,B 0.000,C 90.000,E1 115.668} C_DIS
LIN {X -0.100,Y -218.804,Z 1930.638,A 0.000,B 0.000,C 90.000,E1 114.899} C_DIS
LIN {X 0.041,Y -224.192,Z 1930.621,A 0.000,B 0.000,C 90.000,E1 111.791} C_DIS
LIN {X 0.125,Y -284.143,Z 1930.621,A 0.000,B 0.000,C 90.000,E1 111.770} C_DIS
LIN {X 0.029,Y -285.319,Z 1930.621,A 0.000,B 0.000,C 90.000,E1 111.770} C_DIS
LIN {X 0.001,Y -288.702,Z 1930.620,A 0.000,B 0.000,C 90.000,E1 111.642} C_DIS
LIN {X -0.068,Y -291.971,Z 1930.619,A 0.000,B 0.000,C 90.000,E1 111.408} C_DIS
LIN {X 0.124,Y -295.648,Z 1930.616,A 0.000,B 0.000,C 90.000,E1 110.918} C_DIS
LIN {X -0.064,Y -310.909,Z 1930.602,A 0.000,B 0.000,C 90.000,E1 108.308} C_DIS
LIN {X 0.078,Y -325.637,Z 1930.589,A 0.000,B 0.000,C 90.000,E1 106.024} C_DIS
LIN {X 0.167,Y -339.457,Z 1930.579,A 0.000,B 0.000,C 90.000,E1 104.120} C_DIS
LIN {X 0.025,Y -354.467,Z 1930.568,A 0.000,B 0.000,C 90.000,E1 102.299} C_DIS
LIN {X 0.168,Y -372.937,Z 1930.557,A 0.000,B 0.000,C 90.000,E1 100.254} C_DIS
LIN {X -0.069,Y -391.804,Z 1930.547,A 0.000,B 0.000,C 90.000,E1 98.454} C_DIS
LIN {X -0.052,Y -411.082,Z 1930.538,A 0.000,B 0.000,C 90.000,E1 96.777} C_DIS
LIN {X -0.110,Y -433.488,Z 1930.528,A 0.000,B 0.000,C 90.000,E1 95.049} C_DIS
LIN {X -0.131,Y -439.148,Z 1930.526,A 0.000,B 0.000,C 90.000,E1 94.645} C_DIS
LIN {X -0.142,Y -443.312,Z 1930.523,A 0.000,B 0.000,C 90.000,E1 94.245} C_DIS
LIN {X 0.186,Y -445.031,Z 1930.522,A 0.000,B 0.000,C 90.000,E1 93.955} C_DIS
LIN {X 0.040,Y -446.352,Z 1930.521,A 0.000,B 0.000,C 90.000,E1 93.726} C_DIS
LIN {X -0.036,Y -448.174,Z 1930.518,A 0.000,B 0.000,C 90.000,E1 93.212} C_DIS
LIN {X -0.078,Y -448.934,Z 1930.515,A 0.000,B 0.000,C 90.000,E1 92.694} C_DIS
LIN {X -0.132,Y -448.759,Z 1930.512,A 0.000,B 0.000,C 90.000,E1 92.178} C_DIS
LIN {X -0.165,Y -447.629,Z 1930.509,A 0.000,B 0.000,C 90.000,E1 91.661} C_DIS
LIN {X 0.034,Y -446.655,Z 1930.508,A 0.000,B 0.000,C 90.000,E1 91.375} C_DIS
LIN {X -0.212,Y -445.351,Z 1930.506,A 0.000,B 0.000,C 90.000,E1 91.146} C_DIS
LIN {X 0.163,Y -433.874,Z 1930.496,A 0.000,B 0.000,C 90.000,E1 89.255} C_DIS
LIN {X 0.179,Y -423.849,Z 1930.487,A 0.000,B 0.000,C 90.000,E1 87.650} C_DIS
LIN {X 0.138,Y -412.073,Z 1930.477,A 0.000,B 0.000,C 90.000,E1 85.755} C_DIS
LIN {X -0.196,Y -401.914,Z 1930.467,A 0.000,B 0.000,C 90.000,E1 84.147} C_DIS
LIN {X -0.212,Y -389.929,Z 1930.456,A 0.000,B 0.000,C 90.000,E1 82.186} C_DIS
LIN {X 0.021,Y -378.044,Z 1930.445,A 0.000,B 0.000,C 90.000,E1 80.151} C_DIS
LIN {X 0.035,Y -363.052,Z 1930.431,A 0.000,B 0.000,C 90.000,E1 77.521} C_DIS
LIN {X 0.105,Y -345.856,Z 1930.412,A 0.000,B 0.000,C 90.000,E1 74.212} C_DIS
LIN {X 0.048,Y -333.920,Z 1930.399,A 0.000,B 0.000,C 90.000,E1 71.764} C_DIS
LIN {X 0.057,Y -323.675,Z 1930.387,A 0.000,B 0.000,C 90.000,E1 69.571} C_DIS
LIN {X 0.147,Y -309.617,Z 1930.369,A 0.000,B 0.000,C 90.000,E1 66.357} C_DIS
LIN {X -0.003,Y -300.141,Z 1930.356,A 0.000,B 0.000,C 90.000,E1 64.101} C_DIS
LIN {X -0.123,Y -288.103,Z 1930.339,A 0.000,B 0.000,C 90.000,E1 61.129} C_DIS
LIN {X -0.024,Y -280.038,Z 1930.328,A 0.000,B 0.000,C 90.000,E1 59.076} C_DIS
LIN {X 0.148,Y -270.508,Z 1930.315,A 0.000,B 0.000,C 90.000,E1 56.628} C_DIS
LIN {X 0.063,Y -263.662,Z 1930.305,A 0.000,B 0.000,C 90.000,E1 54.895} C_DIS
LIN {X -0.046,Y -254.034,Z 1930.291,A 0.000,B 0.000,C 90.000,E1 52.431} C_DIS
LIN {X -0.102,Y -244.458,Z 1930.277,A 0.000,B 0.000,C 90.000,E1 49.908} C_DIS
LIN {X 0.087,Y -233.733,Z 1930.261,A 0.000,B 0.000,C 90.000,E1 46.905} C_DIS
LIN {X 0.149,Y -223.421,Z 1930.244,A 0.000,B 0.000,C 90.000,E1 43.866} C_DIS
LIN {X -0.033,Y -213.618,Z 1930.227,A 0.000,B 0.000,C 90.000,E1 40.825} C_DIS
LIN {X -0.121,Y -205.612,Z 1930.211,A 0.000,B 0.000,C 90.000,E1 38.096} C_DIS
LIN {X -0.009,Y -197.318,Z 1930.194,A 0.000,B 0.000,C 90.000,E1 34.865} C_DIS
LIN {X 0.046,Y -189.758,Z 1930.176,A 0.000,B 0.000,C 90.000,E1 31.592} C_DIS
LIN {X 0.044,Y -182.952,Z 1930.157,A 0.000,B 0.000,C 90.000,E1 28.281} C_DIS
LIN {X -0.055,Y -176.843,Z 1930.139,A 0.000,B 0.000,C 90.000,E1 24.951} C_DIS
LIN {X -0.032,Y -171.567,Z 1930.120,A 0.000,B 0.000,C 90.000,E1 21.535} C_DIS
LIN {X 0.057,Y -167.078,Z 1930.100,A 0.000,B 0.000,C 90.000,E1 18.055} C_DIS
LIN {X -0.013,Y -163.438,Z 1930.081,A 0.000,B 0.000,C 90.000,E1 14.592} C_DIS
LIN {X -0.026,Y -159.726,Z 1930.057,A 0.000,B 0.000,C 90.000,E1 10.197} C_DIS
LIN {X 0.035,Y -157.166,Z 1930.032,A 0.000,B 0.000,C 90.000,E1 5.739} C_DIS
LIN {X -0.028,Y -154.883,Z 1929.997,A 0.000,B 0.000,C 90.000,E1 359.542} C_DIS
LIN {X -0.004,Y -154.209,Z 1929.948,A 0.000,B 0.000,C 90.000,E1 350.557} C_DIS
LIN {X 0.003,Y -156.197,Z 1929.908,A 0.000,B 0.000,C 90.000,E1 343.378} C_DIS
LIN {X 0.039,Y -158.576,Z 1929.883,A 0.000,B 0.000,C 90.000,E1 338.901} C_DIS
LIN {X 0.054,Y -162.172,Z 1929.858,A 0.000,B 0.000,C 90.000,E1 334.460} C_DIS
LIN {X -0.039,Y -166.052,Z 1929.839,A 0.000,B 0.000,C 90.000,E1 330.973} C_DIS
LIN {X 0.057,Y -170.929,Z 1929.819,A 0.000,B 0.000,C 90.000,E1 327.454} C_DIS
LIN {X -0.031,Y -175.225,Z 1929.805,A 0.000,B 0.000,C 90.000,E1 324.895} C_DIS
LIN {X 0.022,Y -180.189,Z 1929.791,A 0.000,B 0.000,C 90.000,E1 322.316} C_DIS
LIN {X 0.021,Y -186.048,Z 1929.777,A 0.000,B 0.000,C 90.000,E1 319.784} C_DIS
LIN {X -0.014,Y -191.658,Z 1929.765,A 0.000,B 0.000,C 90.000,E1 317.715} C_DIS
LIN {X 0.023,Y -199.325,Z 1929.751,A 0.000,B 0.000,C 90.000,E1 315.243} C_DIS
LIN {X -0.076,Y -207.914,Z 1929.738,A 0.000,B 0.000,C 90.000,E1 312.852} C_DIS
LIN {X -0.096,Y -218.976,Z 1929.723,A 0.000,B 0.000,C 90.000,E1 310.092} C_DIS
LIN {X -0.031,Y -232.901,Z 1929.705,A 0.000,B 0.000,C 90.000,E1 306.996} C_DIS
LIN {X 0.031,Y -247.963,Z 1929.689,A 0.000,B 0.000,C 90.000,E1 303.992} C_DIS
LIN {X 0.081,Y -259.886,Z 1929.677,A 0.000,B 0.000,C 90.000,E1 301.799} C_DIS
LIN {X 0.086,Y -271.950,Z 1929.665,A 0.000,B 0.000,C 90.000,E1 299.667} C_DIS
LIN {X -0.141,Y -281.842,Z 1929.655,A 0.000,B 0.000,C 90.000,E1 297.975} C_DIS
LIN {X 0.031,Y -291.443,Z 1929.646,A 0.000,B 0.000,C 90.000,E1 296.232} C_DIS
LIN {X 0.110,Y -296.861,Z 1929.640,A 0.000,B 0.000,C 90.000,E1 295.207} C_DIS
LIN {X 0.113,Y -301.665,Z 1929.635,A 0.000,B 0.000,C 90.000,E1 294.207} C_DIS
LIN {X -0.002,Y -304.470,Z 1929.631,A 0.000,B 0.000,C 90.000,E1 293.567} C_DIS
LIN {X 0.059,Y -306.874,Z 1929.627,A 0.000,B 0.000,C 90.000,E1 292.898} C_DIS
LIN {X -0.026,Y -308.886,Z 1929.624,A 0.000,B 0.000,C 90.000,E1 292.259} C_DIS
LIN {X 0.061,Y -310.558,Z 1929.620,A 0.000,B 0.000,C 90.000,E1 291.589} C_DIS
LIN {X -0.125,Y -311.901,Z 1929.616,A 0.000,B 0.000,C 90.000,E1 290.972} C_DIS
LIN {X -0.010,Y -312.903,Z 1929.613,A 0.000,B 0.000,C 90.000,E1 290.301} C_DIS
LIN {X 0.114,Y -313.542,Z 1929.609,A 0.000,B 0.000,C 90.000,E1 289.631} C_DIS
LIN {X -0.155,Y -313.885,Z 1929.606,A 0.000,B 0.000,C 90.000,E1 289.033} C_DIS
LIN {X -0.019,Y -313.876,Z 1929.602,A 0.000,B 0.000,C 90.000,E1 288.362} C_DIS
LIN {X 0.115,Y -313.489,Z 1929.598,A 0.000,B 0.000,C 90.000,E1 287.692} C_DIS
LIN {X -0.144,Y -312.677,Z 1929.595,A 0.000,B 0.000,C 90.000,E1 287.094} C_DIS
LIN {X -0.106,Y -311.382,Z 1929.591,A 0.000,B 0.000,C 90.000,E1 286.441} C_DIS
LIN {X -0.070,Y -309.535,Z 1929.588,A 0.000,B 0.000,C 90.000,E1 285.788} C_DIS
LIN {X -0.042,Y -307.083,Z 1929.584,A 0.000,B 0.000,C 90.000,E1 285.134} C_DIS
LIN {X -0.034,Y -303.848,Z 1929.580,A 0.000,B 0.000,C 90.000,E1 284.481} C_DIS
LIN {X -0.077,Y -296.118,Z 1929.573,A 0.000,B 0.000,C 90.000,E1 283.175} C_DIS
LIN {X 0.015,Y -290.860,Z 1929.568,A 0.000,B 0.000,C 90.000,E1 282.187} C_DIS
LIN {X -0.077,Y -286.506,Z 1929.564,A 0.000,B 0.000,C 90.000,E1 281.535} C_DIS
LIN {X 0.027,Y -281.162,Z 1929.560,A 0.000,B 0.000,C 90.000,E1 280.838} C_DIS
LIN {X 0.024,Y -274.921,Z 1929.557,A 0.000,B 0.000,C 90.000,E1 280.197} C_DIS
LIN {X 0.075,Y -268.479,Z 1929.553,A 0.000,B 0.000,C 90.000,E1 279.613} C_DIS
LIN {X -0.138,Y -261.841,Z 1929.551,A 0.000,B 0.000,C 90.000,E1 279.151} C_DIS
LIN {X -0.022,Y -255.119,Z 1929.548,A 0.000,B 0.000,C 90.000,E1 278.681} C_DIS
LIN {X 0.040,Y -248.178,Z 1929.546,A 0.000,B 0.000,C 90.000,E1 278.276} C_DIS
LIN {X 0.095,Y -240.699,Z 1929.544,A 0.000,B 0.000,C 90.000,E1 277.936} C_DIS
LIN {X -0.008,Y -232.673,Z 1929.543,A 0.000,B 0.000,C 90.000,E1 277.701} C_DIS
LIN {X -0.087,Y -221.988,Z 1929.542,A 0.000,B 0.000,C 90.000,E1 277.530} C_DIS
LIN {X -0.022,Y -216.244,Z 1929.542,A 0.000,B 0.000,C 90.000,E1 277.466} C_DIS
LIN {X -0.049,Y -180.197,Z 1929.541,A 0.000,B 0.000,C 90.000,E1 277.466} C_DIS
LIN {X 0.067,Y -181.027,Z 1929.530,A 0.000,B 0.000,C 90.000,E1 275.391} C_DIS
LIN {X 0.042,Y -181.579,Z 1929.502,A 0.000,B 0.000,C 90.000,E1 270.344} C_DIS
LIN {X 0.017,Y -180.904,Z 1929.474,A 0.000,B 0.000,C 90.000,E1 265.298} C_DIS
LIN {X -0.032,Y -180.246,Z 1929.465,A 0.000,B 0.000,C 90.000,E1 263.628} C_DIS
LIN {X -0.014,Y -178.734,Z 1929.441,A 0.000,B 0.000,C 90.000,E1 259.398} C_DIS
LIN {X 0.054,Y -175.782,Z 1929.413,A 0.000,B 0.000,C 90.000,E1 254.283} C_DIS
LIN {X 0.040,Y -171.967,Z 1929.384,A 0.000,B 0.000,C 90.000,E1 249.156} C_DIS
LIN {X 0.078,Y -171.363,Z 1929.380,A 0.000,B 0.000,C 90.000,E1 248.284} C_DIS
LIN {X 0.055,Y -167.612,Z 1929.355,A 0.000,B 0.000,C 90.000,E1 243.973} C_DIS
LIN {X 0.067,Y -166.260,Z 1929.346,A 0.000,B 0.000,C 90.000,E1 242.231} C_DIS
LIN {X 0.055,Y -163.014,Z 1929.326,A 0.000,B 0.000,C 90.000,E1 238.742} C_DIS
LIN {X -0.032,Y -160.937,Z 1929.312,A 0.000,B 0.000,C 90.000,E1 236.135} C_DIS
LIN {X 0.078,Y -157.697,Z 1929.292,A 0.000,B 0.000,C 90.000,E1 232.557} C_DIS
LIN {X 0.015,Y -155.736,Z 1929.277,A 0.000,B 0.000,C 90.000,E1 229.908} C_DIS
LIN {X 0.069,Y -151.994,Z 1929.252,A 0.000,B 0.000,C 90.000,E1 225.405} C_DIS
LIN {X 0.085,Y -150.239,Z 1929.237,A 0.000,B 0.000,C 90.000,E1 222.690} C_DIS
LIN {X 0.008,Y -146.998,Z 1929.212,A 0.000,B 0.000,C 90.000,E1 218.177} C_DIS
LIN {X -0.003,Y -145.584,Z 1929.197,A 0.000,B 0.000,C 90.000,E1 215.438} C_DIS
LIN {X -0.008,Y -142.971,Z 1929.171,A 0.000,B 0.000,C 90.000,E1 210.846} C_DIS
LIN {X 0.044,Y -141.598,Z 1929.151,A 0.000,B 0.000,C 90.000,E1 207.129} C_DIS
LIN {X -0.039,Y -139.422,Z 1929.115,A 0.000,B 0.000,C 90.000,E1 200.663} C_DIS
LIN {X 0.011,Y -139.150,Z 1929.104,A 0.000,B 0.000,C 90.000,E1 198.779} C_DIS
LIN {X 0.034,Y -138.345,Z 1929.058,A 0.000,B 0.000,C 90.000,E1 190.366} C_DIS
LIN {X 0.019,Y -139.486,Z 1929.006,A 0.000,B 0.000,C 90.000,E1 181.031} C_DIS
LIN {X -0.041,Y -141.086,Z 1928.975,A 0.000,B 0.000,C 90.000,E1 175.469} C_DIS
LIN {X 0.055,Y -142.463,Z 1928.959,A 0.000,B 0.000,C 90.000,E1 172.648} C_DIS
LIN {X 0.003,Y -144.708,Z 1928.934,A 0.000,B 0.000,C 90.000,E1 168.049} C_DIS
LIN {X -0.046,Y -147.306,Z 1928.913,A 0.000,B 0.000,C 90.000,E1 164.393} C_DIS
LIN {X -0.031,Y -150.626,Z 1928.888,A 0.000,B 0.000,C 90.000,E1 159.826} C_DIS
LIN {X 0.045,Y -154.101,Z 1928.868,A 0.000,B 0.000,C 90.000,E1 156.177} C_DIS
LIN {X -0.031,Y -157.525,Z 1928.848,A 0.000,B 0.000,C 90.000,E1 152.615} C_DIS
LIN {X -0.087,Y -161.760,Z 1928.828,A 0.000,B 0.000,C 90.000,E1 149.076} C_DIS
LIN {X 0.020,Y -165.952,Z 1928.808,A 0.000,B 0.000,C 90.000,E1 145.515} C_DIS
LIN {X 0.016,Y -170.944,Z 1928.789,A 0.000,B 0.000,C 90.000,E1 142.029} C_DIS
LIN {X -0.064,Y -175.813,Z 1928.770,A 0.000,B 0.000,C 90.000,E1 138.609} C_DIS
LIN {X 0.064,Y -181.420,Z 1928.751,A 0.000,B 0.000,C 90.000,E1 135.162} C_DIS
LIN {X -0.062,Y -186.923,Z 1928.732,A 0.000,B 0.000,C 90.000,E1 131.838} C_DIS
LIN {X 0.011,Y -191.502,Z 1928.719,A 0.000,B 0.000,C 90.000,E1 129.322} C_DIS
LIN {X 0.096,Y -197.365,Z 1928.700,A 0.000,B 0.000,C 90.000,E1 126.011} C_DIS
LIN {X 0.021,Y -200.642,Z 1928.691,A 0.000,B 0.000,C 90.000,E1 124.405} C_DIS
LIN {X -0.069,Y -206.526,Z 1928.673,A 0.000,B 0.000,C 90.000,E1 121.209} C_DIS
LIN {X 0.025,Y -209.816,Z 1928.664,A 0.000,B 0.000,C 90.000,E1 119.589} C_DIS
LIN {X -0.049,Y -217.175,Z 1928.643,A 0.000,B 0.000,C 90.000,E1 115.668} C_DIS
LIN {X -0.095,Y -218.801,Z 1928.638,A 0.000,B 0.000,C 90.000,E1 114.899} C_DIS
LIN {X 0.046,Y -224.188,Z 1928.621,A 0.000,B 0.000,C 90.000,E1 111.791} C_DIS
LIN {X 0.132,Y -284.160,Z 1928.621,A 0.000,B 0.000,C 90.000,E1 111.770} C_DIS
LIN {X 0.036,Y -285.323,Z 1928.621,A 0.000,B 0.000,C 90.000,E1 111.770} C_DIS
LIN {X 0.003,Y -288.710,Z 1928.620,A 0.000,B 0.000,C 90.000,E1 111.642} C_DIS
LIN {X -0.070,Y -291.983,Z 1928.619,A 0.000,B 0.000,C 90.000,E1 111.408} C_DIS
LIN {X 0.116,Y -295.660,Z 1928.616,A 0.000,B 0.000,C 90.000,E1 110.918} C_DIS
LIN {X -0.080,Y -310.926,Z 1928.602,A 0.000,B 0.000,C 90.000,E1 108.308} C_DIS
LIN {X 0.061,Y -325.655,Z 1928.589,A 0.000,B 0.000,C 90.000,E1 106.024} C_DIS
LIN {X 0.150,Y -339.478,Z 1928.579,A 0.000,B 0.000,C 90.000,E1 104.120} C_DIS
LIN {X 0.008,Y -354.489,Z 1928.568,A 0.000,B 0.000,C 90.000,E1 102.299} C_DIS
LIN {X 0.152,Y -372.959,Z 1928.557,A 0.000,B 0.000,C 90.000,E1 100.254} C_DIS
LIN {X -0.084,Y -391.827,Z 1928.547,A 0.000,B 0.000,C 90.000,E1 98.454} C_DIS
LIN {X -0.067,Y -411.105,Z 1928.538,A 0.000,B 0.000,C 90.000,E1 96.777} C_DIS
LIN {X -0.124,Y -433.512,Z 1928.528,A 0.000,B 0.000,C 90.000,E1 95.049} C_DIS
LIN {X -0.145,Y -439.170,Z 1928.526,A 0.000,B 0.000,C 90.000,E1 94.645} C_DIS
LIN {X -0.156,Y -443.319,Z 1928.523,A 0.000,B 0.000,C 90.000,E1 94.245} C_DIS
LIN {X 0.168,Y -445.037,Z 1928.522,A 0.000,B 0.000,C 90.000,E1 93.955} C_DIS
LIN {X 0.015,Y -446.356,Z 1928.521,A 0.000,B 0.000,C 90.000,E1 93.726} C_DIS
LIN {X -0.059,Y -448.169,Z 1928.518,A 0.000,B 0.000,C 90.000,E1 93.212} C_DIS
LIN {X -0.102,Y -448.922,Z 1928.515,A 0.000,B 0.000,C 90.000,E1 92.694} C_DIS
LIN {X -0.156,Y -448.740,Z 1928.512,A 0.000,B 0.000,C 90.000,E1 92.178} C_DIS
LIN {X -0.189,Y -447.602,Z 1928.509,A 0.000,B 0.000,C 90.000,E1 91.661} C_DIS
LIN {X 0.010,Y -446.624,Z 1928.508,A 0.000,B 0.000,C 90.000,E1 91.375} C_DIS
LIN {X 0.209,Y -445.313,Z 1928.506,A 0.000,B 0.000,C 90.000,E1 91.088} C_DIS
LIN {X 0.138,Y -433.834,Z 1928.496,A 0.000,B 0.000,C 90.000,E1 89.255} C_DIS
LIN {X 0.154,Y -423.809,Z 1928.487,A 0.000,B 0.000,C 90.000,E1 87.650} C_DIS
LIN {X 0.114,Y -412.034,Z 1928.477,A 0.000,B 0.000,C 90.000,E1 85.755} C_DIS
LIN {X 0.179,Y -401.874,Z 1928.467,A 0.000,B 0.000,C 90.000,E1 84.090} C_DIS
LIN {X 0.149,Y -389.889,Z 1928.456,A 0.000,B 0.000,C 90.000,E1 82.129} C_DIS
LIN {X -0.004,Y -378.003,Z 1928.445,A 0.000,B 0.000,C 90.000,E1 80.151} C_DIS
LIN {X 0.010,Y -363.011,Z 1928.431,A 0.000,B 0.000,C 90.000,E1 77.521} C_DIS
LIN {X 0.080,Y -345.816,Z 1928.412,A 0.000,B 0.000,C 90.000,E1 74.212} C_DIS
LIN {X 0.022,Y -333.879,Z 1928.399,A 0.000,B 0.000,C 90.000,E1 71.764} C_DIS
LIN {X 0.031,Y -323.634,Z 1928.387,A 0.000,B 0.000,C 90.000,E1 69.571} C_DIS
LIN {X 0.121,Y -309.577,Z 1928.369,A 0.000,B 0.000,C 90.000,E1 66.357} C_DIS
LIN {X 0.079,Y -301.466,Z 1928.358,A 0.000,B 0.000,C 90.000,E1 64.409} C_DIS
LIN {X 0.003,Y -289.372,Z 1928.341,A 0.000,B 0.000,C 90.000,E1 61.435} C_DIS
LIN {X -0.013,Y -281.347,Z 1928.330,A 0.000,B 0.000,C 90.000,E1 59.410} C_DIS
LIN {X 0.036,Y -271.817,Z 1928.317,A 0.000,B 0.000,C 90.000,E1 56.993} C_DIS
LIN {X 0.037,Y -263.622,Z 1928.305,A 0.000,B 0.000,C 90.000,E1 54.895} C_DIS
LIN {X 0.083,Y -253.996,Z 1928.291,A 0.000,B 0.000,C 90.000,E1 52.396} C_DIS
LIN {X -0.127,Y -244.419,Z 1928.277,A 0.000,B 0.000,C 90.000,E1 49.908} C_DIS
LIN {X 0.062,Y -233.694,Z 1928.261,A 0.000,B 0.000,C 90.000,E1 46.905} C_DIS
LIN {X 0.123,Y -223.381,Z 1928.244,A 0.000,B 0.000,C 90.000,E1 43.866} C_DIS
LIN {X -0.058,Y -213.581,Z 1928.227,A 0.000,B 0.000,C 90.000,E1 40.825} C_DIS
LIN {X 0.016,Y -205.578,Z 1928.211,A 0.000,B 0.000,C 90.000,E1 38.051} C_DIS
LIN {X -0.035,Y -197.288,Z 1928.194,A 0.000,B 0.000,C 90.000,E1 34.865} C_DIS
LIN {X 0.021,Y -189.732,Z 1928.176,A 0.000,B 0.000,C 90.000,E1 31.592} C_DIS
LIN {X 0.021,Y -182.929,Z 1928.157,A 0.000,B 0.000,C 90.000,E1 28.281} C_DIS
LIN {X 0.082,Y -176.823,Z 1928.138,A 0.000,B 0.000,C 90.000,E1 24.899} C_DIS
LIN {X -0.057,Y -171.550,Z 1928.120,A 0.000,B 0.000,C 90.000,E1 21.535} C_DIS
LIN {X 0.033,Y -167.063,Z 1928.100,A 0.000,B 0.000,C 90.000,E1 18.055} C_DIS
LIN {X -0.036,Y -163.422,Z 1928.081,A 0.000,B 0.000,C 90.000,E1 14.592} C_DIS
LIN {X -0.049,Y -159.712,Z 1928.057,A 0.000,B 0.000,C 90.000,E1 10.197} C_DIS
LIN {X 0.011,Y -157.156,Z 1928.032,A 0.000,B 0.000,C 90.000,E1 5.739} C_DIS
LIN {X -0.028,Y -154.874,Z 1927.997,A 0.000,B 0.000,C 90.000,E1 359.542} C_DIS
LIN {X -0.005,Y -154.201,Z 1927.948,A 0.000,B 0.000,C 90.000,E1 350.557} C_DIS
LIN {X 0.003,Y -156.192,Z 1927.908,A 0.000,B 0.000,C 90.000,E1 343.378} C_DIS
LIN {X 0.038,Y -158.573,Z 1927.883,A 0.000,B 0.000,C 90.000,E1 338.901} C_DIS
LIN {X 0.052,Y -162.170,Z 1927.858,A 0.000,B 0.000,C 90.000,E1 334.460} C_DIS
LIN {X -0.041,Y -166.056,Z 1927.839,A 0.000,B 0.000,C 90.000,E1 330.973} C_DIS
LIN {X 0.056,Y -170.933,Z 1927.819,A 0.000,B 0.000,C 90.000,E1 327.454} C_DIS
LIN {X -0.031,Y -175.231,Z 1927.805,A 0.000,B 0.000,C 90.000,E1 324.895} C_DIS
LIN {X 0.021,Y -180.197,Z 1927.791,A 0.000,B 0.000,C 90.000,E1 322.316} C_DIS
LIN {X 0.020,Y -186.056,Z 1927.777,A 0.000,B 0.000,C 90.000,E1 319.784} C_DIS
LIN {X -0.015,Y -191.667,Z 1927.765,A 0.000,B 0.000,C 90.000,E1 317.715} C_DIS
LIN {X 0.023,Y -199.331,Z 1927.751,A 0.000,B 0.000,C 90.000,E1 315.243} C_DIS
LIN {X -0.076,Y -207.920,Z 1927.738,A 0.000,B 0.000,C 90.000,E1 312.852} C_DIS
LIN {X -0.096,Y -218.984,Z 1927.723,A 0.000,B 0.000,C 90.000,E1 310.092} C_DIS
LIN {X -0.031,Y -232.911,Z 1927.705,A 0.000,B 0.000,C 90.000,E1 306.996} C_DIS
LIN {X 0.031,Y -247.973,Z 1927.689,A 0.000,B 0.000,C 90.000,E1 303.992} C_DIS
LIN {X 0.081,Y -259.895,Z 1927.677,A 0.000,B 0.000,C 90.000,E1 301.799} C_DIS
LIN {X 0.086,Y -271.959,Z 1927.665,A 0.000,B 0.000,C 90.000,E1 299.667} C_DIS
LIN {X -0.141,Y -281.850,Z 1927.655,A 0.000,B 0.000,C 90.000,E1 297.975} C_DIS
LIN {X 0.031,Y -291.451,Z 1927.646,A 0.000,B 0.000,C 90.000,E1 296.232} C_DIS
LIN {X 0.112,Y -296.873,Z 1927.640,A 0.000,B 0.000,C 90.000,E1 295.207} C_DIS
LIN {X 0.113,Y -301.678,Z 1927.635,A 0.000,B 0.000,C 90.000,E1 294.207} C_DIS
LIN {X -0.002,Y -304.481,Z 1927.631,A 0.000,B 0.000,C 90.000,E1 293.567} C_DIS
LIN {X 0.060,Y -306.885,Z 1927.627,A 0.000,B 0.000,C 90.000,E1 292.898} C_DIS
LIN {X -0.025,Y -308.900,Z 1927.624,A 0.000,B 0.000,C 90.000,E1 292.259} C_DIS
LIN {X 0.063,Y -310.572,Z 1927.620,A 0.000,B 0.000,C 90.000,E1 291.589} C_DIS
LIN {X -0.123,Y -311.914,Z 1927.616,A 0.000,B 0.000,C 90.000,E1 290.972} C_DIS
LIN {X -0.009,Y -312.917,Z 1927.613,A 0.000,B 0.000,C 90.000,E1 290.301} C_DIS
LIN {X 0.115,Y -313.556,Z 1927.609,A 0.000,B 0.000,C 90.000,E1 289.631} C_DIS
LIN {X -0.153,Y -313.900,Z 1927.606,A 0.000,B 0.000,C 90.000,E1 289.033} C_DIS
LIN {X -0.017,Y -313.891,Z 1927.602,A 0.000,B 0.000,C 90.000,E1 288.362} C_DIS
LIN {X 0.117,Y -313.504,Z 1927.598,A 0.000,B 0.000,C 90.000,E1 287.692} C_DIS
LIN {X -0.143,Y -312.692,Z 1927.595,A 0.000,B 0.000,C 90.000,E1 287.094} C_DIS
LIN {X -0.104,Y -311.402,Z 1927.591,A 0.000,B 0.000,C 90.000,E1 286.441} C_DIS
LIN {X -0.069,Y -309.551,Z 1927.588,A 0.000,B 0.000,C 90.000,E1 285.788} C_DIS
LIN {X -0.041,Y -307.101,Z 1927.584,A 0.000,B 0.000,C 90.000,E1 285.134} C_DIS
LIN {X -0.032,Y -303.866,Z 1927.580,A 0.000,B 0.000,C 90.000,E1 284.481} C_DIS
LIN {X -0.074,Y -296.139,Z 1927.573,A 0.000,B 0.000,C 90.000,E1 283.175} C_DIS
LIN {X 0.019,Y -290.873,Z 1927.568,A 0.000,B 0.000,C 90.000,E1 282.187} C_DIS
LIN {X -0.073,Y -286.522,Z 1927.564,A 0.000,B 0.000,C 90.000,E1 281.535} C_DIS
LIN {X 0.032,Y -281.175,Z 1927.560,A 0.000,B 0.000,C 90.000,E1 280.838} C_DIS
LIN {X 0.029,Y -274.928,Z 1927.557,A 0.000,B 0.000,C 90.000,E1 280.197} C_DIS
LIN {X 0.078,Y -268.487,Z 1927.553,A 0.000,B 0.000,C 90.000,E1 279.613} C_DIS
LIN {X -0.135,Y -261.852,Z 1927.551,A 0.000,B 0.000,C 90.000,E1 279.151} C_DIS
LIN {X -0.016,Y -255.132,Z 1927.548,A 0.000,B 0.000,C 90.000,E1 278.681} C_DIS
LIN {X 0.045,Y -248.194,Z 1927.546,A 0.000,B 0.000,C 90.000,E1 278.276} C_DIS
LIN {X 0.100,Y -240.713,Z 1927.544,A 0.000,B 0.000,C 90.000,E1 277.936} C_DIS
LIN {X -0.003,Y -232.688,Z 1927.543,A 0.000,B 0.000,C 90.000,E1 277.701} C_DIS
LIN {X -0.082,Y -222.005,Z 1927.542,A 0.000,B 0.000,C 90.000,E1 277.530} C_DIS
LIN {X -0.018,Y -216.266,Z 1927.542,A 0.000,B 0.000,C 90.000,E1 277.466} C_DIS
LIN {X -0.045,Y -180.197,Z 1927.541,A 0.000,B 0.000,C 90.000,E1 277.466} C_DIS
LIN {X 0.071,Y -181.027,Z 1927.530,A 0.000,B 0.000,C 90.000,E1 275.391} C_DIS
LIN {X 0.046,Y -181.579,Z 1927.502,A 0.000,B 0.000,C 90.000,E1 270.344} C_DIS
LIN {X 0.021,Y -180.904,Z 1927.474,A 0.000,B 0.000,C 90.000,E1 265.298} C_DIS
LIN {X -0.029,Y -180.247,Z 1927.465,A 0.000,B 0.000,C 90.000,E1 263.628} C_DIS
LIN {X -0.010,Y -178.735,Z 1927.441,A 0.000,B 0.000,C 90.000,E1 259.398} C_DIS
LIN {X 0.057,Y -175.783,Z 1927.413,A 0.000,B 0.000,C 90.000,E1 254.283} C_DIS
LIN {X 0.045,Y -171.967,Z 1927.384,A 0.000,B 0.000,C 90.000,E1 249.156} C_DIS
LIN {X 0.082,Y -171.365,Z 1927.380,A 0.000,B 0.000,C 90.000,E1 248.284} C_DIS
LIN {X -0.092,Y -167.612,Z 1927.355,A 0.000,B 0.000,C 90.000,E1 244.024} C_DIS
LIN {X 0.071,Y -166.261,Z 1927.346,A 0.000,B 0.000,C 90.000,E1 242.231} C_DIS
LIN {X 0.059,Y -163.015,Z 1927.326,A 0.000,B 0.000,C 90.000,E1 238.742} C_DIS
LIN {X -0.029,Y -160.939,Z 1927.312,A 0.000,B 0.000,C 90.000,E1 236.135} C_DIS
LIN {X 0.081,Y -157.698,Z 1927.292,A 0.000,B 0.000,C 90.000,E1 232.557} C_DIS
LIN {X 0.019,Y -155.737,Z 1927.277,A 0.000,B 0.000,C 90.000,E1 229.908} C_DIS
LIN {X 0.073,Y -151.995,Z 1927.252,A 0.000,B 0.000,C 90.000,E1 225.405} C_DIS
LIN {X 0.088,Y -150.240,Z 1927.237,A 0.000,B 0.000,C 90.000,E1 222.690} C_DIS
LIN {X 0.011,Y -146.999,Z 1927.212,A 0.000,B 0.000,C 90.000,E1 218.177} C_DIS
LIN {X 0.001,Y -145.584,Z 1927.197,A 0.000,B 0.000,C 90.000,E1 215.438} C_DIS
LIN {X -0.005,Y -142.972,Z 1927.171,A 0.000,B 0.000,C 90.000,E1 210.846} C_DIS
LIN {X 0.048,Y -141.599,Z 1927.151,A 0.000,B 0.000,C 90.000,E1 207.129} C_DIS
LIN {X -0.036,Y -139.422,Z 1927.115,A 0.000,B 0.000,C 90.000,E1 200.663} C_DIS
LIN {X 0.015,Y -139.150,Z 1927.104,A 0.000,B 0.000,C 90.000,E1 198.779} C_DIS
LIN {X 0.037,Y -138.345,Z 1927.058,A 0.000,B 0.000,C 90.000,E1 190.366} C_DIS
LIN {X 0.023,Y -139.486,Z 1927.006,A 0.000,B 0.000,C 90.000,E1 181.031} C_DIS
LIN {X -0.037,Y -141.086,Z 1926.975,A 0.000,B 0.000,C 90.000,E1 175.469} C_DIS
LIN {X 0.058,Y -142.463,Z 1926.959,A 0.000,B 0.000,C 90.000,E1 172.648} C_DIS
LIN {X 0.006,Y -144.707,Z 1926.934,A 0.000,B 0.000,C 90.000,E1 168.049} C_DIS
LIN {X -0.042,Y -147.304,Z 1926.913,A 0.000,B 0.000,C 90.000,E1 164.393} C_DIS
LIN {X -0.028,Y -150.624,Z 1926.888,A 0.000,B 0.000,C 90.000,E1 159.826} C_DIS
LIN {X 0.049,Y -154.101,Z 1926.868,A 0.000,B 0.000,C 90.000,E1 156.177} C_DIS
LIN {X -0.028,Y -157.523,Z 1926.848,A 0.000,B 0.000,C 90.000,E1 152.615} C_DIS
LIN {X -0.083,Y -161.758,Z 1926.828,A 0.000,B 0.000,C 90.000,E1 149.076} C_DIS
LIN {X 0.023,Y -165.950,Z 1926.808,A 0.000,B 0.000,C 90.000,E1 145.515} C_DIS
LIN {X 0.020,Y -170.942,Z 1926.789,A 0.000,B 0.000,C 90.000,E1 142.029} C_DIS
LIN {X -0.059,Y -175.811,Z 1926.770,A 0.000,B 0.000,C 90.000,E1 138.609} C_DIS
LIN {X 0.067,Y -181.418,Z 1926.751,A 0.000,B 0.000,C 90.000,E1 135.162} C_DIS
LIN {X -0.057,Y -186.921,Z 1926.732,A 0.000,B 0.000,C 90.000,E1 131.838} C_DIS
LIN {X 0.015,Y -191.500,Z 1926.719,A 0.000,B 0.000,C 90.000,E1 129.322} C_DIS
LIN {X 0.100,Y -197.363,Z 1926.700,A 0.000,B 0.000,C 90.000,E1 126.011} C_DIS
LIN {X 0.025,Y -200.639,Z 1926.691,A 0.000,B 0.000,C 90.000,E1 124.405} C_DIS
LIN {X -0.065,Y -206.523,Z 1926.673,A 0.000,B 0.000,C 90.000,E1 121.209} C_DIS
LIN {X 0.029,Y -209.814,Z 1926.664,A 0.000,B 0.000,C 90.000,E1 119.589} C_DIS
LIN {X -0.044,Y -217.172,Z 1926.643,A 0.000,B 0.000,C 90.000,E1 115.668} C_DIS
LIN {X -0.091,Y -218.798,Z 1926.638,A 0.000,B 0.000,C 90.000,E1 114.899} C_DIS
LIN {X 0.050,Y -224.187,Z 1926.621,A 0.000,B 0.000,C 90.000,E1 111.791} C_DIS
LIN {X 0.137,Y -284.190,Z 1926.621,A 0.000,B 0.000,C 90.000,E1 111.770} C_DIS
LIN {X 0.041,Y -285.333,Z 1926.621,A 0.000,B 0.000,C 90.000,E1 111.770} C_DIS
LIN {X 0.003,Y -288.728,Z 1926.620,A 0.000,B 0.000,C 90.000,E1 111.642} C_DIS
LIN {X -0.078,Y -292.006,Z 1926.619,A 0.000,B 0.000,C 90.000,E1 111.408} C_DIS
LIN {X 0.097,Y -295.683,Z 1926.616,A 0.000,B 0.000,C 90.000,E1 110.918} C_DIS
LIN {X -0.110,Y -310.958,Z 1926.602,A 0.000,B 0.000,C 90.000,E1 108.308} C_DIS
LIN {X 0.031,Y -325.691,Z 1926.589,A 0.000,B 0.000,C 90.000,E1 106.024} C_DIS
LIN {X 0.119,Y -339.516,Z 1926.579,A 0.000,B 0.000,C 90.000,E1 104.120} C_DIS
LIN {X -0.024,Y -354.532,Z 1926.568,A 0.000,B 0.000,C 90.000,E1 102.299} C_DIS
LIN {X 0.121,Y -373.003,Z 1926.557,A 0.000,B 0.000,C 90.000,E1 100.254} C_DIS
LIN {X -0.114,Y -391.871,Z 1926.547,A 0.000,B 0.000,C 90.000,E1 98.454} C_DIS
LIN {X -0.094,Y -411.150,Z 1926.538,A 0.000,B 0.000,C 90.000,E1 96.777} C_DIS
LIN {X -0.151,Y -433.559,Z 1926.528,A 0.000,B 0.000,C 90.000,E1 95.049} C_DIS
LIN {X -0.172,Y -439.215,Z 1926.526,A 0.000,B 0.000,C 90.000,E1 94.645} C_DIS
LIN {X -0.184,Y -443.339,Z 1926.523,A 0.000,B 0.000,C 90.000,E1 94.245} C_DIS
LIN {X 0.132,Y -445.055,Z 1926.522,A 0.000,B 0.000,C 90.000,E1 93.955} C_DIS
LIN {X -0.028,Y -446.371,Z 1926.521,A 0.000,B 0.000,C 90.000,E1 93.726} C_DIS
LIN {X -0.102,Y -448.168,Z 1926.518,A 0.000,B 0.000,C 90.000,E1 93.212} C_DIS
LIN {X -0.146,Y -448.910,Z 1926.515,A 0.000,B 0.000,C 90.000,E1 92.694} C_DIS
LIN {X -0.199,Y -448.718,Z 1926.512,A 0.000,B 0.000,C 90.000,E1 92.178} C_DIS
LIN {X 0.215,Y -447.566,Z 1926.509,A 0.000,B 0.000,C 90.000,E1 91.604} C_DIS
LIN {X -0.033,Y -446.582,Z 1926.508,A 0.000,B 0.000,C 90.000,E1 91.375} C_DIS
LIN {X 0.166,Y -445.262,Z 1926.506,A 0.000,B 0.000,C 90.000,E1 91.088} C_DIS
LIN {X 0.096,Y -433.779,Z 1926.496,A 0.000,B 0.000,C 90.000,E1 89.255} C_DIS
LIN {X 0.111,Y -423.754,Z 1926.487,A 0.000,B 0.000,C 90.000,E1 87.650} C_DIS
LIN {X 0.070,Y -411.979,Z 1926.476,A 0.000,B 0.000,C 90.000,E1 85.755} C_DIS
LIN {X 0.136,Y -401.819,Z 1926.467,A 0.000,B 0.000,C 90.000,E1 84.090} C_DIS
LIN {X 0.107,Y -389.834,Z 1926.456,A 0.000,B 0.000,C 90.000,E1 82.129} C_DIS
LIN {X -0.046,Y -377.948,Z 1926.445,A 0.000,B 0.000,C 90.000,E1 80.151} C_DIS
LIN {X -0.032,Y -362.955,Z 1926.431,A 0.000,B 0.000,C 90.000,E1 77.521} C_DIS
LIN {X 0.038,Y -345.763,Z 1926.412,A 0.000,B 0.000,C 90.000,E1 74.212} C_DIS
LIN {X -0.019,Y -333.826,Z 1926.399,A 0.000,B 0.000,C 90.000,E1 71.764} C_DIS
LIN {X -0.010,Y -323.581,Z 1926.386,A 0.000,B 0.000,C 90.000,E1 69.571} C_DIS
LIN {X 0.079,Y -309.525,Z 1926.369,A 0.000,B 0.000,C 90.000,E1 66.357} C_DIS
LIN {X 0.038,Y -301.413,Z 1926.358,A 0.000,B 0.000,C 90.000,E1 64.409} C_DIS
LIN {X -0.039,Y -289.317,Z 1926.341,A 0.000,B 0.000,C 90.000,E1 61.435} C_DIS
LIN {X -0.054,Y -281.289,Z 1926.330,A 0.000,B 0.000,C 90.000,E1 59.410} C_DIS
LIN {X -0.006,Y -271.764,Z 1926.317,A 0.000,B 0.000,C 90.000,E1 56.993} C_DIS
LIN {X -0.003,Y -263.569,Z 1926.305,A 0.000,B 0.000,C 90.000,E1 54.895} C_DIS
LIN {X 0.042,Y -253.945,Z 1926.291,A 0.000,B 0.000,C 90.000,E1 52.396} C_DIS
LIN {X 0.020,Y -244.367,Z 1926.277,A 0.000,B 0.000,C 90.000,E1 49.865} C_DIS
LIN {X 0.023,Y -233.643,Z 1926.261,A 0.000,B 0.000,C 90.000,E1 46.905} C_DIS
LIN {X 0.086,Y -223.329,Z 1926.244,A 0.000,B 0.000,C 90.000,E1 43.866} C_DIS
LIN {X 0.066,Y -213.532,Z 1926.227,A 0.000,B 0.000,C 90.000,E1 40.782} C_DIS
LIN {X 0.105,Y -205.534,Z 1926.211,A 0.000,B 0.000,C 90.000,E1 38.016} C_DIS
LIN {X 0.090,Y -197.248,Z 1926.194,A 0.000,B 0.000,C 90.000,E1 34.818} C_DIS
LIN {X -0.015,Y -189.698,Z 1926.176,A 0.000,B 0.000,C 90.000,E1 31.592} C_DIS
LIN {X -0.015,Y -182.898,Z 1926.157,A 0.000,B 0.000,C 90.000,E1 28.281} C_DIS
LIN {X 0.046,Y -176.797,Z 1926.138,A 0.000,B 0.000,C 90.000,E1 24.899} C_DIS
LIN {X -0.092,Y -171.526,Z 1926.120,A 0.000,B 0.000,C 90.000,E1 21.535} C_DIS
LIN {X -0.003,Y -167.043,Z 1926.100,A 0.000,B 0.000,C 90.000,E1 18.055} C_DIS
LIN {X -0.071,Y -163.404,Z 1926.081,A 0.000,B 0.000,C 90.000,E1 14.592} C_DIS
LIN {X -0.083,Y -159.696,Z 1926.057,A 0.000,B 0.000,C 90.000,E1 10.197} C_DIS
LIN {X -0.023,Y -157.142,Z 1926.032,A 0.000,B 0.000,C 90.000,E1 5.739} C_DIS
LIN {X -0.028,Y -154.865,Z 1925.997,A 0.000,B 0.000,C 90.000,E1 359.542} C_DIS
LIN {X -0.006,Y -154.195,Z 1925.948,A 0.000,B 0.000,C 90.000,E1 350.557} C_DIS
LIN {X 0.002,Y -156.187,Z 1925.908,A 0.000,B 0.000,C 90.000,E1 343.378} C_DIS
LIN {X 0.037,Y -158.570,Z 1925.883,A 0.000,B 0.000,C 90.000,E1 338.901} C_DIS
LIN {X 0.052,Y -162.168,Z 1925.858,A 0.000,B 0.000,C 90.000,E1 334.460} C_DIS
LIN {X -0.042,Y -166.058,Z 1925.839,A 0.000,B 0.000,C 90.000,E1 330.973} C_DIS
LIN {X 0.055,Y -170.938,Z 1925.819,A 0.000,B 0.000,C 90.000,E1 327.454} C_DIS
LIN {X -0.032,Y -175.238,Z 1925.805,A 0.000,B 0.000,C 90.000,E1 324.895} C_DIS
LIN {X 0.020,Y -180.206,Z 1925.791,A 0.000,B 0.000,C 90.000,E1 322.316} C_DIS
LIN {X 0.019,Y -186.065,Z 1925.777,A 0.000,B 0.000,C 90.000,E1 319.784} C_DIS
LIN {X -0.015,Y -191.676,Z 1925.765,A 0.000,B 0.000,C 90.000,E1 317.715} C_DIS
LIN {X 0.022,Y -199.337,Z 1925.751,A 0.000,B 0.000,C 90.000,E1 315.243} C_DIS
LIN {X -0.077,Y -207.927,Z 1925.738,A 0.000,B 0.000,C 90.000,E1 312.852} C_DIS
LIN {X -0.096,Y -218.992,Z 1925.723,A 0.000,B 0.000,C 90.000,E1 310.092} C_DIS
LIN {X -0.032,Y -232.920,Z 1925.705,A 0.000,B 0.000,C 90.000,E1 306.996} C_DIS
LIN {X 0.031,Y -247.984,Z 1925.689,A 0.000,B 0.000,C 90.000,E1 303.992} C_DIS
LIN {X 0.081,Y -259.905,Z 1925.677,A 0.000,B 0.000,C 90.000,E1 301.799} C_DIS
LIN {X 0.087,Y -271.968,Z 1925.665,A 0.000,B 0.000,C 90.000,E1 299.667} C_DIS
LIN {X -0.140,Y -281.858,Z 1925.655,A 0.000,B 0.000,C 90.000,E1 297.975} C_DIS
LIN {X 0.033,Y -291.459,Z 1925.646,A 0.000,B 0.000,C 90.000,E1 296.232} C_DIS
LIN {X 0.113,Y -296.884,Z 1925.640,A 0.000,B 0.000,C 90.000,E1 295.207} C_DIS
LIN {X 0.115,Y -301.692,Z 1925.635,A 0.000,B 0.000,C 90.000,E1 294.207} C_DIS
LIN {X 0.000,Y -304.493,Z 1925.631,A 0.000,B 0.000,C 90.000,E1 293.567} C_DIS
LIN {X 0.062,Y -306.897,Z 1925.627,A 0.000,B 0.000,C 90.000,E1 292.898} C_DIS
LIN {X -0.024,Y -308.912,Z 1925.624,A 0.000,B 0.000,C 90.000,E1 292.259} C_DIS
LIN {X 0.065,Y -310.586,Z 1925.620,A 0.000,B 0.000,C 90.000,E1 291.589} C_DIS
LIN {X -0.122,Y -311.927,Z 1925.616,A 0.000,B 0.000,C 90.000,E1 290.972} C_DIS
LIN {X -0.007,Y -312.932,Z 1925.613,A 0.000,B 0.000,C 90.000,E1 290.301} C_DIS
LIN {X 0.118,Y -313.571,Z 1925.609,A 0.000,B 0.000,C 90.000,E1 289.631} C_DIS
LIN {X -0.151,Y -313.914,Z 1925.606,A 0.000,B 0.000,C 90.000,E1 289.033} C_DIS
LIN {X -0.016,Y -313.905,Z 1925.602,A 0.000,B 0.000,C 90.000,E1 288.362} C_DIS
LIN {X 0.119,Y -313.518,Z 1925.598,A 0.000,B 0.000,C 90.000,E1 287.692} C_DIS
LIN {X -0.141,Y -312.706,Z 1925.595,A 0.000,B 0.000,C 90.000,E1 287.094} C_DIS
LIN {X -0.101,Y -311.421,Z 1925.591,A 0.000,B 0.000,C 90.000,E1 286.441} C_DIS
LIN {X -0.066,Y -309.568,Z 1925.588,A 0.000,B 0.000,C 90.000,E1 285.788} C_DIS
LIN {X -0.039,Y -307.119,Z 1925.584,A 0.000,B 0.000,C 90.000,E1 285.134} C_DIS
LIN {X -0.029,Y -303.884,Z 1925.580,A 0.000,B 0.000,C 90.000,E1 284.481} C_DIS
LIN {X -0.072,Y -296.160,Z 1925.573,A 0.000,B 0.000,C 90.000,E1 283.175} C_DIS
LIN {X 0.023,Y -290.887,Z 1925.568,A 0.000,B 0.000,C 90.000,E1 282.187} C_DIS
LIN {X -0.069,Y -286.538,Z 1925.564,A 0.000,B 0.000,C 90.000,E1 281.535} C_DIS
LIN {X 0.036,Y -281.189,Z 1925.560,A 0.000,B 0.000,C 90.000,E1 280.838} C_DIS
LIN {X 0.033,Y -274.934,Z 1925.557,A 0.000,B 0.000,C 90.000,E1 280.197} C_DIS
LIN {X 0.080,Y -268.495,Z 1925.553,A 0.000,B 0.000,C 90.000,E1 279.613} C_DIS
LIN {X -0.131,Y -261.861,Z 1925.551,A 0.000,B 0.000,C 90.000,E1 279.151} C_DIS
LIN {X -0.011,Y -255.145,Z 1925.548,A 0.000,B 0.000,C 90.000,E1 278.681} C_DIS
LIN {X 0.051,Y -248.208,Z 1925.546,A 0.000,B 0.000,C 90.000,E1 278.276} C_DIS
LIN {X 0.105,Y -240.725,Z 1925.544,A 0.000,B 0.000,C 90.000,E1 277.936} C_DIS
LIN {X 0.003,Y -232.691,Z 1925.543,A 0.000,B 0.000,C 90.000,E1 277.701} C_DIS
LIN {X -0.078,Y -222.016,Z 1925.542,A 0.000,B 0.000,C 90.000,E1 277.530} C_DIS
LIN {X -0.014,Y -216.271,Z 1925.542,A 0.000,B 0.000,C 90.000,E1 277.466} C_DIS
LIN {X -0.042,Y -180.197,Z 1925.541,A 0.000,B 0.000,C 90.000,E1 277.466} C_DIS
LIN {X 0.074,Y -181.027,Z 1925.530,A 0.000,B 0.000,C 90.000,E1 275.391} C_DIS
LIN {X 0.049,Y -181.579,Z 1925.502,A 0.000,B 0.000,C 90.000,E1 270.344} C_DIS
LIN {X 0.025,Y -180.904,Z 1925.474,A 0.000,B 0.000,C 90.000,E1 265.298} C_DIS
LIN {X -0.025,Y -180.247,Z 1925.465,A 0.000,B 0.000,C 90.000,E1 263.628} C_DIS
LIN {X -0.006,Y -178.735,Z 1925.441,A 0.000,B 0.000,C 90.000,E1 259.398} C_DIS
LIN {X 0.060,Y -175.783,Z 1925.413,A 0.000,B 0.000,C 90.000,E1 254.283} C_DIS
LIN {X 0.048,Y -171.967,Z 1925.384,A 0.000,B 0.000,C 90.000,E1 249.156} C_DIS
LIN {X 0.085,Y -171.366,Z 1925.380,A 0.000,B 0.000,C 90.000,E1 248.284} C_DIS
LIN {X -0.089,Y -167.614,Z 1925.355,A 0.000,B 0.000,C 90.000,E1 244.024} C_DIS
LIN {X 0.074,Y -166.263,Z 1925.346,A 0.000,B 0.000,C 90.000,E1 242.231} C_DIS
LIN {X 0.061,Y -163.015,Z 1925.326,A 0.000,B 0.000,C 90.000,E1 238.742} C_DIS
LIN {X -0.025,Y -160.940,Z 1925.312,A 0.000,B 0.000,C 90.000,E1 236.135} C_DIS
LIN {X 0.085,Y -157.699,Z 1925.292,A 0.000,B 0.000,C 90.000,E1 232.557} C_DIS
LIN {X 0.022,Y -155.738,Z 1925.277,A 0.000,B 0.000,C 90.000,E1 229.908} C_DIS
LIN {X 0.076,Y -151.996,Z 1925.252,A 0.000,B 0.000,C 90.000,E1 225.405} C_DIS
LIN {X 0.091,Y -150.241,Z 1925.237,A 0.000,B 0.000,C 90.000,E1 222.690} C_DIS
LIN {X 0.015,Y -147.000,Z 1925.212,A 0.000,B 0.000,C 90.000,E1 218.177} C_DIS
LIN {X 0.004,Y -145.585,Z 1925.197,A 0.000,B 0.000,C 90.000,E1 215.438} C_DIS
LIN {X -0.002,Y -142.973,Z 1925.171,A 0.000,B 0.000,C 90.000,E1 210.846} C_DIS
LIN {X 0.051,Y -141.600,Z 1925.151,A 0.000,B 0.000,C 90.000,E1 207.129} C_DIS
LIN {X -0.033,Y -139.422,Z 1925.115,A 0.000,B 0.000,C 90.000,E1 200.663} C_DIS
LIN {X 0.017,Y -139.151,Z 1925.104,A 0.000,B 0.000,C 90.000,E1 198.779} C_DIS
LIN {X 0.040,Y -138.345,Z 1925.058,A 0.000,B 0.000,C 90.000,E1 190.366} C_DIS
LIN {X 0.026,Y -139.486,Z 1925.006,A 0.000,B 0.000,C 90.000,E1 181.031} C_DIS
LIN {X -0.034,Y -141.086,Z 1924.975,A 0.000,B 0.000,C 90.000,E1 175.469} C_DIS
LIN {X 0.060,Y -142.462,Z 1924.959,A 0.000,B 0.000,C 90.000,E1 172.648} C_DIS
LIN {X 0.009,Y -144.706,Z 1924.934,A 0.000,B 0.000,C 90.000,E1 168.049} C_DIS
LIN {X -0.039,Y -147.304,Z 1924.913,A 0.000,B 0.000,C 90.000,E1 164.393} C_DIS
LIN {X -0.025,Y -150.624,Z 1924.888,A 0.000,B 0.000,C 90.000,E1 159.826} C_DIS
LIN {X 0.052,Y -154.100,Z 1924.868,A 0.000,B 0.000,C 90.000,E1 156.177} C_DIS
LIN {X -0.024,Y -157.522,Z 1924.848,A 0.000,B 0.000,C 90.000,E1 152.615} C_DIS
LIN {X -0.080,Y -161.756,Z 1924.828,A 0.000,B 0.000,C 90.000,E1 149.076} C_DIS
LIN {X 0.026,Y -165.949,Z 1924.808,A 0.000,B 0.000,C 90.000,E1 145.515} C_DIS
LIN {X 0.023,Y -170.941,Z 1924.789,A 0.000,B 0.000,C 90.000,E1 142.029} C_DIS
LIN {X -0.056,Y -175.809,Z 1924.770,A 0.000,B 0.000,C 90.000,E1 138.609} C_DIS
LIN {X 0.071,Y -181.416,Z 1924.751,A 0.000,B 0.000,C 90.000,E1 135.162} C_DIS
LIN {X -0.054,Y -186.919,Z 1924.732,A 0.000,B 0.000,C 90.000,E1 131.838} C_DIS
LIN {X 0.019,Y -191.498,Z 1924.719,A 0.000,B 0.000,C 90.000,E1 129.322} C_DIS
LIN {X 0.104,Y -197.361,Z 1924.700,A 0.000,B 0.000,C 90.000,E1 126.011} C_DIS
LIN {X 0.028,Y -200.637,Z 1924.691,A 0.000,B 0.000,C 90.000,E1 124.405} C_DIS
LIN {X -0.062,Y -206.521,Z 1924.673,A 0.000,B 0.000,C 90.000,E1 121.209} C_DIS
LIN {X 0.033,Y -209.811,Z 1924.664,A 0.000,B 0.000,C 90.000,E1 119.589} C_DIS
LIN {X -0.041,Y -217.170,Z 1924.643,A 0.000,B 0.000,C 90.000,E1 115.668} C_DIS
LIN {X -0.087,Y -218.797,Z 1924.638,A 0.000,B 0.000,C 90.000,E1 114.899} C_DIS
LIN {X -0.128,Y -224.173,Z 1924.621,A 0.000,B 0.000,C 90.000,E1 111.844} C_DIS
LIN {X 0.069,Y -283.376,Z 1924.621,A 0.000,B 0.000,C 90.000,E1 111.791} C_DIS
LIN {X 0.046,Y -285.350,Z 1924.621,A 0.000,B 0.000,C 90.000,E1 111.770} C_DIS
LIN {X 0.043,Y -288.215,Z 1924.620,A 0.000,B 0.000,C 90.000,E1 111.663} C_DIS
LIN {X 0.146,Y -291.540,Z 1924.619,A 0.000,B 0.000,C 90.000,E1 111.408} C_DIS
LIN {X -0.075,Y -295.196,Z 1924.617,A 0.000,B 0.000,C 90.000,E1 111.025} C_DIS
LIN {X -0.149,Y -300.707,Z 1924.611,A 0.000,B 0.000,C 90.000,E1 110.066} C_DIS
LIN {X -0.155,Y -314.390,Z 1924.599,A 0.000,B 0.000,C 90.000,E1 107.764} C_DIS
LIN {X 0.061,Y -329.475,Z 1924.586,A 0.000,B 0.000,C 90.000,E1 105.481} C_DIS
LIN {X 0.136,Y -343.629,Z 1924.576,A 0.000,B 0.000,C 90.000,E1 103.592} C_DIS
LIN {X 0.105,Y -358.956,Z 1924.565,A 0.000,B 0.000,C 90.000,E1 101.771} C_DIS
LIN {X 0.126,Y -377.540,Z 1924.555,A 0.000,B 0.000,C 90.000,E1 99.792} C_DIS
LIN {X 0.179,Y -396.503,Z 1924.545,A 0.000,B 0.000,C 90.000,E1 97.992} C_DIS
LIN {X 0.122,Y -418.638,Z 1924.534,A 0.000,B 0.000,C 90.000,E1 96.144} C_DIS
LIN {X -0.139,Y -438.355,Z 1924.526,A 0.000,B 0.000,C 90.000,E1 94.702} C_DIS
LIN {X -0.130,Y -442.808,Z 1924.524,A 0.000,B 0.000,C 90.000,E1 94.302} C_DIS
LIN {X -0.211,Y -445.920,Z 1924.521,A 0.000,B 0.000,C 90.000,E1 93.841} C_DIS
LIN {X -0.033,Y -447.081,Z 1924.520,A 0.000,B 0.000,C 90.000,E1 93.555} C_DIS
LIN {X 0.147,Y -447.931,Z 1924.518,A 0.000,B 0.000,C 90.000,E1 93.269} C_DIS
LIN {X 0.108,Y -448.837,Z 1924.515,A 0.000,B 0.000,C 90.000,E1 92.751} C_DIS
LIN {X 0.054,Y -448.801,Z 1924.512,A 0.000,B 0.000,C 90.000,E1 92.236} C_DIS
LIN {X 0.019,Y -447.821,Z 1924.510,A 0.000,B 0.000,C 90.000,E1 91.718} C_DIS
LIN {X -0.029,Y -445.738,Z 1924.507,A 0.000,B 0.000,C 90.000,E1 91.203} C_DIS
LIN {X 0.193,Y -435.970,Z 1924.498,A 0.000,B 0.000,C 90.000,E1 89.599} C_DIS
LIN {X -0.181,Y -426.012,Z 1924.489,A 0.000,B 0.000,C 90.000,E1 88.051} C_DIS
LIN {X -0.073,Y -412.538,Z 1924.477,A 0.000,B 0.000,C 90.000,E1 85.869} C_DIS
LIN {X 0.007,Y -402.386,Z 1924.468,A 0.000,B 0.000,C 90.000,E1 84.204} C_DIS
LIN {X -0.003,Y -390.404,Z 1924.457,A 0.000,B 0.000,C 90.000,E1 82.243} C_DIS
LIN {X -0.202,Y -378.505,Z 1924.446,A 0.000,B 0.000,C 90.000,E1 80.274} C_DIS
LIN {X -0.156,Y -365.126,Z 1924.433,A 0.000,B 0.000,C 90.000,E1 77.937} C_DIS
LIN {X -0.043,Y -349.314,Z 1924.416,A 0.000,B 0.000,C 90.000,E1 74.936} C_DIS
LIN {X -0.027,Y -335.792,Z 1924.401,A 0.000,B 0.000,C 90.000,E1 72.181} C_DIS
LIN {X -0.119,Y -324.055,Z 1924.387,A 0.000,B 0.000,C 90.000,E1 69.699} C_DIS
LIN {X -0.013,Y -309.967,Z 1924.369,A 0.000,B 0.000,C 90.000,E1 66.485} C_DIS
LIN {X -0.021,Y -300.494,Z 1924.357,A 0.000,B 0.000,C 90.000,E1 64.204} C_DIS
LIN {X 0.136,Y -288.434,Z 1924.340,A 0.000,B 0.000,C 90.000,E1 61.179} C_DIS
LIN {X -0.145,Y -280.375,Z 1924.329,A 0.000,B 0.000,C 90.000,E1 59.203} C_DIS
LIN {X 0.041,Y -270.858,Z 1924.315,A 0.000,B 0.000,C 90.000,E1 56.755} C_DIS
LIN {X -0.119,Y -262.632,Z 1924.304,A 0.000,B 0.000,C 90.000,E1 54.689} C_DIS
LIN {X -0.096,Y -253.026,Z 1924.290,A 0.000,B 0.000,C 90.000,E1 52.190} C_DIS
LIN {X 0.024,Y -243.442,Z 1924.276,A 0.000,B 0.000,C 90.000,E1 49.622} C_DIS
LIN {X 0.009,Y -232.770,Z 1924.259,A 0.000,B 0.000,C 90.000,E1 46.662} C_DIS
LIN {X 0.050,Y -222.478,Z 1924.242,A 0.000,B 0.000,C 90.000,E1 43.623} C_DIS
LIN {X -0.082,Y -211.553,Z 1924.223,A 0.000,B 0.000,C 90.000,E1 40.172} C_DIS
LIN {X 0.078,Y -203.729,Z 1924.208,A 0.000,B 0.000,C 90.000,E1 37.363} C_DIS
LIN {X -0.086,Y -195.599,Z 1924.190,A 0.000,B 0.000,C 90.000,E1 34.199} C_DIS
LIN {X -0.064,Y -188.218,Z 1924.172,A 0.000,B 0.000,C 90.000,E1 30.924} C_DIS
LIN {X -0.025,Y -181.562,Z 1924.153,A 0.000,B 0.000,C 90.000,E1 27.590} C_DIS
LIN {X 0.010,Y -175.626,Z 1924.135,A 0.000,B 0.000,C 90.000,E1 24.207} C_DIS
LIN {X 0.002,Y -170.511,Z 1924.115,A 0.000,B 0.000,C 90.000,E1 20.791} C_DIS
LIN {X 0.008,Y -166.228,Z 1924.096,A 0.000,B 0.000,C 90.000,E1 17.330} C_DIS
LIN {X 0.033,Y -162.724,Z 1924.077,A 0.000,B 0.000,C 90.000,E1 13.828} C_DIS
LIN {X 0.020,Y -159.796,Z 1924.057,A 0.000,B 0.000,C 90.000,E1 10.310} C_DIS
LIN {X 0.078,Y -157.205,Z 1924.033,A 0.000,B 0.000,C 90.000,E1 5.853} C_DIS
LIN {X 0.000,Y -154.982,Z 1924.000,A 0.000,B 0.000,C 90.000,E1 360.000} C_DIS
LIN {X 0.055,Y -154.113,Z 1923.953,A 0.000,B 0.000,C 90.000,E1 351.432} C_DIS
LIN {X -0.026,Y -155.842,Z 1923.913,A 0.000,B 0.000,C 90.000,E1 344.283} C_DIS
LIN {X 0.036,Y -158.568,Z 1923.883,A 0.000,B 0.000,C 90.000,E1 338.901} C_DIS
LIN {X 0.051,Y -162.166,Z 1923.858,A 0.000,B 0.000,C 90.000,E1 334.460} C_DIS
LIN {X -0.043,Y -166.061,Z 1923.839,A 0.000,B 0.000,C 90.000,E1 330.973} C_DIS
LIN {X 0.054,Y -170.942,Z 1923.819,A 0.000,B 0.000,C 90.000,E1 327.454} C_DIS
LIN {X -0.034,Y -175.244,Z 1923.805,A 0.000,B 0.000,C 90.000,E1 324.895} C_DIS
LIN {X 0.019,Y -180.214,Z 1923.791,A 0.000,B 0.000,C 90.000,E1 322.316} C_DIS
LIN {X 0.018,Y -186.074,Z 1923.777,A 0.000,B 0.000,C 90.000,E1 319.784} C_DIS
LIN {X -0.017,Y -191.685,Z 1923.765,A 0.000,B 0.000,C 90.000,E1 317.715} C_DIS
LIN {X 0.022,Y -199.343,Z 1923.751,A 0.000,B 0.000,C 90.000,E1 315.243} C_DIS
LIN {X -0.076,Y -207.934,Z 1923.738,A 0.000,B 0.000,C 90.000,E1 312.852} C_DIS
LIN {X -0.098,Y -219.000,Z 1923.723,A 0.000,B 0.000,C 90.000,E1 310.092} C_DIS
LIN {X -0.032,Y -232.930,Z 1923.705,A 0.000,B 0.000,C 90.000,E1 306.996} C_DIS
LIN {X 0.031,Y -247.993,Z 1923.689,A 0.000,B 0.000,C 90.000,E1 303.992} C_DIS
LIN {X 0.082,Y -259.915,Z 1923.677,A 0.000,B 0.000,C 90.000,E1 301.799} C_DIS
LIN {X 0.086,Y -271.977,Z 1923.665,A 0.000,B 0.000,C 90.000,E1 299.667} C_DIS
LIN {X -0.139,Y -281.867,Z 1923.655,A 0.000,B 0.000,C 90.000,E1 297.975} C_DIS
LIN {X 0.033,Y -291.467,Z 1923.646,A 0.000,B 0.000,C 90.000,E1 296.232} C_DIS
LIN {X 0.114,Y -296.896,Z 1923.640,A 0.000,B 0.000,C 90.000,E1 295.207} C_DIS
LIN {X 0.116,Y -301.704,Z 1923.635,A 0.000,B 0.000,C 90.000,E1 294.207} C_DIS
LIN {X 0.002,Y -304.504,Z 1923.631,A 0.000,B 0.000,C 90.000,E1 293.567} C_DIS
LIN {X 0.063,Y -306.908,Z 1923.627,A 0.000,B 0.000,C 90.000,E1 292.898} C_DIS
LIN {X -0.023,Y -308.924,Z 1923.624,A 0.000,B 0.000,C 90.000,E1 292.259} C_DIS
LIN {X 0.066,Y -310.598,Z 1923.620,A 0.000,B 0.000,C 90.000,E1 291.589} C_DIS
LIN {X -0.120,Y -311.940,Z 1923.616,A 0.000,B 0.000,C 90.000,E1 290.972} C_DIS
LIN {X -0.005,Y -312.947,Z 1923.613,A 0.000,B 0.000,C 90.000,E1 290.301} C_DIS
LIN {X 0.119,Y -313.585,Z 1923.609,A 0.000,B 0.000,C 90.000,E1 289.631} C_DIS
LIN {X -0.149,Y -313.929,Z 1923.606,A 0.000,B 0.000,C 90.000,E1 289.033} C_DIS
LIN {X -0.014,Y -313.920,Z 1923.602,A 0.000,B 0.000,C 90.000,E1 288.362} C_DIS
LIN {X 0.121,Y -313.533,Z 1923.598,A 0.000,B 0.000,C 90.000,E1 287.692} C_DIS
LIN {X -0.138,Y -312.722,Z 1923.595,A 0.000,B 0.000,C 90.000,E1 287.094} C_DIS
LIN {X -0.099,Y -311.439,Z 1923.591,A 0.000,B 0.000,C 90.000,E1 286.441} C_DIS
LIN {X -0.064,Y -309.585,Z 1923.588,A 0.000,B 0.000,C 90.000,E1 285.788} C_DIS
LIN {X -0.036,Y -307.137,Z 1923.584,A 0.000,B 0.000,C 90.000,E1 285.134} C_DIS
LIN {X -0.027,Y -303.905,Z 1923.580,A 0.000,B 0.000,C 90.000,E1 284.481} C_DIS
LIN {X -0.069,Y -296.181,Z 1923.573,A 0.000,B 0.000,C 90.000,E1 283.175} C_DIS
LIN {X 0.015,Y -293.843,Z 1923.571,A 0.000,B 0.000,C 90.000,E1 282.715} C_DIS
LIN {X 0.037,Y -341.645,Z 1923.571,A 0.000,B 0.000,C 90.000,E1 282.703} C_DIS
LIN {X -0.051,Y -343.601,Z 1923.570,A 0.000,B 0.000,C 90.000,E1 282.535} C_DIS
LIN {X -0.007,Y -345.754,Z 1923.567,A 0.000,B 0.000,C 90.000,E1 282.007} C_DIS
LIN {X -0.183,Y -346.822,Z 1923.563,A 0.000,B 0.000,C 90.000,E1 281.422} C_DIS
LIN {X -0.005,Y -346.672,Z 1923.560,A 0.000,B 0.000,C 90.000,E1 280.782} C_DIS
LIN {X -0.161,Y -345.680,Z 1923.557,A 0.000,B 0.000,C 90.000,E1 280.197} C_DIS
LIN {X 0.116,Y -343.160,Z 1923.553,A 0.000,B 0.000,C 90.000,E1 279.443} C_DIS
LIN {X -0.026,Y -341.530,Z 1923.551,A 0.000,B 0.000,C 90.000,E1 279.208} C_DIS
LIN {X 0.093,Y -339.648,Z 1923.550,A 0.000,B 0.000,C 90.000,E1 279.029} C_DIS
LIN {X 0.033,Y -339.331,Z 1923.550,A 0.000,B 0.000,C 90.000,E1 279.029} C_DIS
LIN {X -0.021,Y -260.471,Z 1923.550,A 0.000,B 0.000,C 90.000,E1 279.029} C_DIS
LIN {X 0.119,Y -252.754,Z 1923.547,A 0.000,B 0.000,C 90.000,E1 278.511} C_DIS
LIN {X 0.022,Y -245.665,Z 1923.545,A 0.000,B 0.000,C 90.000,E1 278.163} C_DIS
LIN {X -0.039,Y -238.044,Z 1923.544,A 0.000,B 0.000,C 90.000,E1 277.871} C_DIS
LIN {X -0.080,Y -229.231,Z 1923.542,A 0.000,B 0.000,C 90.000,E1 277.644} C_DIS
LIN {X 0.036,Y -218.144,Z 1923.542,A 0.000,B 0.000,C 90.000,E1 277.466} C_DIS
LIN {X -0.004,Y -216.503,Z 1923.542,A 0.000,B 0.000,C 90.000,E1 277.466} C_DIS
LIN {X -0.036,Y -180.196,Z 1923.541,A 0.000,B 0.000,C 90.000,E1 277.466} C_DIS
LIN {X -0.072,Y -181.025,Z 1923.530,A 0.000,B 0.000,C 90.000,E1 275.448} C_DIS
LIN {X 0.083,Y -181.578,Z 1923.502,A 0.000,B 0.000,C 90.000,E1 270.344} C_DIS
LIN {X 0.058,Y -180.905,Z 1923.474,A 0.000,B 0.000,C 90.000,E1 265.298} C_DIS
LIN {X 0.008,Y -180.252,Z 1923.465,A 0.000,B 0.000,C 90.000,E1 263.628} C_DIS
LIN {X 0.027,Y -178.742,Z 1923.441,A 0.000,B 0.000,C 90.000,E1 259.398} C_DIS
LIN {X -0.076,Y -175.790,Z 1923.413,A 0.000,B 0.000,C 90.000,E1 254.338} C_DIS
LIN {X -0.080,Y -171.974,Z 1923.384,A 0.000,B 0.000,C 90.000,E1 249.209} C_DIS
LIN {X -0.042,Y -171.376,Z 1923.380,A 0.000,B 0.000,C 90.000,E1 248.337} C_DIS
LIN {X -0.056,Y -167.622,Z 1923.356,A 0.000,B 0.000,C 90.000,E1 244.024} C_DIS
LIN {X -0.041,Y -166.274,Z 1923.346,A 0.000,B 0.000,C 90.000,E1 242.281} C_DIS
LIN {X -0.047,Y -163.024,Z 1923.327,A 0.000,B 0.000,C 90.000,E1 238.791} C_DIS
LIN {X 0.006,Y -160.951,Z 1923.312,A 0.000,B 0.000,C 90.000,E1 236.135} C_DIS
LIN {X -0.010,Y -157.708,Z 1923.292,A 0.000,B 0.000,C 90.000,E1 232.603} C_DIS
LIN {X 0.053,Y -155.747,Z 1923.277,A 0.000,B 0.000,C 90.000,E1 229.908} C_DIS
LIN {X -0.001,Y -152.004,Z 1923.252,A 0.000,B 0.000,C 90.000,E1 225.445} C_DIS
LIN {X -0.091,Y -150.249,Z 1923.237,A 0.000,B 0.000,C 90.000,E1 222.771} C_DIS
LIN {X 0.044,Y -147.006,Z 1923.212,A 0.000,B 0.000,C 90.000,E1 218.177} C_DIS
LIN {X 0.033,Y -145.590,Z 1923.197,A 0.000,B 0.000,C 90.000,E1 215.438} C_DIS
LIN {X -0.046,Y -142.978,Z 1923.171,A 0.000,B 0.000,C 90.000,E1 210.875} C_DIS
LIN {X 0.080,Y -141.605,Z 1923.151,A 0.000,B 0.000,C 90.000,E1 207.129} C_DIS
LIN {X -0.004,Y -139.425,Z 1923.115,A 0.000,B 0.000,C 90.000,E1 200.663} C_DIS
LIN {X 0.046,Y -139.153,Z 1923.104,A 0.000,B 0.000,C 90.000,E1 198.779} C_DIS
LIN {X 0.068,Y -138.344,Z 1923.058,A 0.000,B 0.000,C 90.000,E1 190.366} C_DIS
LIN {X 0.054,Y -139.484,Z 1923.006,A 0.000,B 0.000,C 90.000,E1 181.031} C_DIS
LIN {X -0.005,Y -141.080,Z 1922.975,A 0.000,B 0.000,C 90.000,E1 175.469} C_DIS
LIN {X -0.051,Y -142.457,Z 1922.959,A 0.000,B 0.000,C 90.000,E1 172.704} C_DIS
LIN {X 0.039,Y -144.699,Z 1922.934,A 0.000,B 0.000,C 90.000,E1 168.049} C_DIS
LIN {X -0.010,Y -147.294,Z 1922.913,A 0.000,B 0.000,C 90.000,E1 164.393} C_DIS
LIN {X 0.006,Y -150.614,Z 1922.888,A 0.000,B 0.000,C 90.000,E1 159.826} C_DIS
LIN {X -0.059,Y -154.088,Z 1922.868,A 0.000,B 0.000,C 90.000,E1 156.230} C_DIS
LIN {X 0.007,Y -157.510,Z 1922.848,A 0.000,B 0.000,C 90.000,E1 152.615} C_DIS
LIN {X -0.047,Y -161.742,Z 1922.828,A 0.000,B 0.000,C 90.000,E1 149.076} C_DIS
LIN {X 0.059,Y -165.935,Z 1922.808,A 0.000,B 0.000,C 90.000,E1 145.515} C_DIS
LIN {X -0.049,Y -170.924,Z 1922.789,A 0.000,B 0.000,C 90.000,E1 142.065} C_DIS
LIN {X -0.023,Y -175.792,Z 1922.770,A 0.000,B 0.000,C 90.000,E1 138.609} C_DIS
LIN {X -0.023,Y -181.401,Z 1922.751,A 0.000,B 0.000,C 90.000,E1 135.202} C_DIS
LIN {X -0.020,Y -186.900,Z 1922.732,A 0.000,B 0.000,C 90.000,E1 131.838} C_DIS
LIN {X -0.068,Y -191.481,Z 1922.719,A 0.000,B 0.000,C 90.000,E1 129.358} C_DIS
LIN {X -0.136,Y -197.341,Z 1922.700,A 0.000,B 0.000,C 90.000,E1 126.091} C_DIS
LIN {X 0.064,Y -200.618,Z 1922.691,A 0.000,B 0.000,C 90.000,E1 124.405} C_DIS
LIN {X -0.025,Y -206.501,Z 1922.673,A 0.000,B 0.000,C 90.000,E1 121.209} C_DIS
LIN {X -0.034,Y -209.789,Z 1922.664,A 0.000,B 0.000,C 90.000,E1 119.617} C_DIS
LIN {X -0.004,Y -217.150,Z 1922.643,A 0.000,B 0.000,C 90.000,E1 115.668} C_DIS
LIN {X -0.050,Y -218.776,Z 1922.638,A 0.000,B 0.000,C 90.000,E1 114.899} C_DIS
LIN {X 0.065,Y -224.180,Z 1922.621,A 0.000,B 0.000,C 90.000,E1 111.791} C_DIS
LIN {X 0.052,Y -284.103,Z 1922.621,A 0.000,B 0.000,C 90.000,E1 111.791} C_DIS
LIN {X 0.055,Y -288.193,Z 1922.620,A 0.000,B 0.000,C 90.000,E1 111.663} C_DIS
LIN {X -0.051,Y -291.386,Z 1922.619,A 0.000,B 0.000,C 90.000,E1 111.461} C_DIS
LIN {X -0.081,Y -295.064,Z 1922.617,A 0.000,B 0.000,C 90.000,E1 111.046} C_DIS
LIN {X -0.159,Y -298.711,Z 1922.613,A 0.000,B 0.000,C 90.000,E1 110.429} C_DIS
LIN {X 0.187,Y -312.181,Z 1922.600,A 0.000,B 0.000,C 90.000,E1 108.055} C_DIS
LIN {X -0.049,Y -327.048,Z 1922.588,A 0.000,B 0.000,C 90.000,E1 105.843} C_DIS
LIN {X 0.060,Y -340.992,Z 1922.578,A 0.000,B 0.000,C 90.000,E1 103.939} C_DIS
LIN {X -0.065,Y -356.142,Z 1922.567,A 0.000,B 0.000,C 90.000,E1 102.119} C_DIS
LIN {X 0.143,Y -374.618,Z 1922.556,A 0.000,B 0.000,C 90.000,E1 100.084} C_DIS
LIN {X 0.051,Y -393.558,Z 1922.546,A 0.000,B 0.000,C 90.000,E1 98.276} C_DIS
LIN {X 0.200,Y -415.633,Z 1922.536,A 0.000,B 0.000,C 90.000,E1 96.372} C_DIS
LIN {X -0.012,Y -438.118,Z 1922.526,A 0.000,B 0.000,C 90.000,E1 94.702} C_DIS
LIN {X -0.004,Y -442.662,Z 1922.524,A 0.000,B 0.000,C 90.000,E1 94.302} C_DIS
LIN {X -0.037,Y -445.796,Z 1922.521,A 0.000,B 0.000,C 90.000,E1 93.841} C_DIS
LIN {X 0.141,Y -446.985,Z 1922.520,A 0.000,B 0.000,C 90.000,E1 93.555} C_DIS
LIN {X -0.127,Y -447.858,Z 1922.518,A 0.000,B 0.000,C 90.000,E1 93.326} C_DIS
LIN {X -0.166,Y -448.804,Z 1922.516,A 0.000,B 0.000,C 90.000,E1 92.808} C_DIS
LIN {X -0.222,Y -448.805,Z 1922.513,A 0.000,B 0.000,C 90.000,E1 92.293} C_DIS
LIN {X 0.192,Y -447.866,Z 1922.510,A 0.000,B 0.000,C 90.000,E1 91.718} C_DIS
LIN {X 0.142,Y -445.834,Z 1922.507,A 0.000,B 0.000,C 90.000,E1 91.203} C_DIS
LIN {X 0.189,Y -437.735,Z 1922.500,A 0.000,B 0.000,C 90.000,E1 89.885} C_DIS
LIN {X -0.167,Y -427.810,Z 1922.491,A 0.000,B 0.000,C 90.000,E1 88.339} C_DIS
LIN {X -0.124,Y -416.013,Z 1922.480,A 0.000,B 0.000,C 90.000,E1 86.445} C_DIS
LIN {X 0.115,Y -404.210,Z 1922.469,A 0.000,B 0.000,C 90.000,E1 84.489} C_DIS
LIN {X 0.100,Y -392.252,Z 1922.459,A 0.000,B 0.000,C 90.000,E1 82.534} C_DIS
LIN {X -0.010,Y -380.314,Z 1922.448,A 0.000,B 0.000,C 90.000,E1 80.557} C_DIS
LIN {X 0.019,Y -368.546,Z 1922.436,A 0.000,B 0.000,C 90.000,E1 78.522} C_DIS
LIN {X -0.109,Y -352.495,Z 1922.420,A 0.000,B 0.000,C 90.000,E1 75.574} C_DIS
LIN {X -0.090,Y -338.854,Z 1922.405,A 0.000,B 0.000,C 90.000,E1 72.834} C_DIS
LIN {X 0.101,Y -327.078,Z 1922.391,A 0.000,B 0.000,C 90.000,E1 70.315} C_DIS
LIN {X -0.051,Y -314.198,Z 1922.375,A 0.000,B 0.000,C 90.000,E1 67.486} C_DIS
LIN {X -0.071,Y -303.304,Z 1922.360,A 0.000,B 0.000,C 90.000,E1 64.897} C_DIS
LIN {X 0.037,Y -291.159,Z 1922.344,A 0.000,B 0.000,C 90.000,E1 61.897} C_DIS
LIN {X 0.052,Y -283.164,Z 1922.333,A 0.000,B 0.000,C 90.000,E1 59.871} C_DIS
LIN {X 0.146,Y -273.658,Z 1922.319,A 0.000,B 0.000,C 90.000,E1 57.454} C_DIS
LIN {X 0.032,Y -265.496,Z 1922.308,A 0.000,B 0.000,C 90.000,E1 55.388} C_DIS
LIN {X 0.000,Y -254.493,Z 1922.292,A 0.000,B 0.000,C 90.000,E1 52.557} C_DIS
LIN {X -0.043,Y -244.905,Z 1922.278,A 0.000,B 0.000,C 90.000,E1 50.033} C_DIS
LIN {X 0.002,Y -234.157,Z 1922.261,A 0.000,B 0.000,C 90.000,E1 47.067} C_DIS
LIN {X 0.078,Y -223.829,Z 1922.245,A 0.000,B 0.000,C 90.000,E1 44.028} C_DIS
LIN {X -0.090,Y -213.995,Z 1922.228,A 0.000,B 0.000,C 90.000,E1 40.987} C_DIS
LIN {X -0.038,Y -205.966,Z 1922.212,A 0.000,B 0.000,C 90.000,E1 38.222} C_DIS
LIN {X -0.039,Y -197.644,Z 1922.195,A 0.000,B 0.000,C 90.000,E1 35.025} C_DIS
LIN {X 0.031,Y -190.056,Z 1922.176,A 0.000,B 0.000,C 90.000,E1 31.750} C_DIS
LIN {X 0.045,Y -183.223,Z 1922.158,A 0.000,B 0.000,C 90.000,E1 28.437} C_DIS
LIN {X 0.036,Y -177.080,Z 1922.139,A 0.000,B 0.000,C 90.000,E1 25.079} C_DIS
LIN {X 0.062,Y -171.768,Z 1922.120,A 0.000,B 0.000,C 90.000,E1 21.663} C_DIS
LIN {X -0.003,Y -167.243,Z 1922.101,A 0.000,B 0.000,C 90.000,E1 18.236} C_DIS
LIN {X -0.065,Y -163.563,Z 1922.082,A 0.000,B 0.000,C 90.000,E1 14.773} C_DIS
LIN {X -0.041,Y -159.812,Z 1922.057,A 0.000,B 0.000,C 90.000,E1 10.366} C_DIS
LIN {X 0.016,Y -157.213,Z 1922.033,A 0.000,B 0.000,C 90.000,E1 5.910} C_DIS
LIN {X 0.000,Y -154.974,Z 1922.000,A 0.000,B 0.000,C 90.000,E1 360.000} C_DIS
LIN {X 0.055,Y -154.107,Z 1921.953,A 0.000,B 0.000,C 90.000,E1 351.432} C_DIS
LIN {X -0.026,Y -155.837,Z 1921.913,A 0.000,B 0.000,C 90.000,E1 344.283} C_DIS
LIN {X 0.035,Y -158.566,Z 1921.883,A 0.000,B 0.000,C 90.000,E1 338.901} C_DIS
LIN {X 0.049,Y -162.165,Z 1921.858,A 0.000,B 0.000,C 90.000,E1 334.460} C_DIS
LIN {X -0.044,Y -166.064,Z 1921.839,A 0.000,B 0.000,C 90.000,E1 330.973} C_DIS
LIN {X 0.053,Y -170.948,Z 1921.819,A 0.000,B 0.000,C 90.000,E1 327.454} C_DIS
LIN {X -0.035,Y -175.250,Z 1921.805,A 0.000,B 0.000,C 90.000,E1 324.895} C_DIS
LIN {X 0.018,Y -180.223,Z 1921.791,A 0.000,B 0.000,C 90.000,E1 322.316} C_DIS
LIN {X 0.018,Y -186.083,Z 1921.777,A 0.000,B 0.000,C 90.000,E1 319.784} C_DIS
LIN {X -0.016,Y -191.694,Z 1921.765,A 0.000,B 0.000,C 90.000,E1 317.715} C_DIS
LIN {X 0.021,Y -199.349,Z 1921.751,A 0.000,B 0.000,C 90.000,E1 315.243} C_DIS
LIN {X -0.077,Y -207.940,Z 1921.738,A 0.000,B 0.000,C 90.000,E1 312.852} C_DIS
LIN {X -0.098,Y -219.008,Z 1921.723,A 0.000,B 0.000,C 90.000,E1 310.092} C_DIS
LIN {X -0.032,Y -232.938,Z 1921.705,A 0.000,B 0.000,C 90.000,E1 306.996} C_DIS
LIN {X 0.031,Y -248.004,Z 1921.689,A 0.000,B 0.000,C 90.000,E1 303.992} C_DIS
LIN {X 0.082,Y -259.924,Z 1921.677,A 0.000,B 0.000,C 90.000,E1 301.799} C_DIS
LIN {X 0.087,Y -271.985,Z 1921.665,A 0.000,B 0.000,C 90.000,E1 299.667} C_DIS
LIN {X -0.139,Y -281.876,Z 1921.655,A 0.000,B 0.000,C 90.000,E1 297.975} C_DIS
LIN {X 0.035,Y -291.476,Z 1921.646,A 0.000,B 0.000,C 90.000,E1 296.232} C_DIS
LIN {X 0.115,Y -296.907,Z 1921.640,A 0.000,B 0.000,C 90.000,E1 295.207} C_DIS
LIN {X 0.117,Y -301.717,Z 1921.635,A 0.000,B 0.000,C 90.000,E1 294.207} C_DIS
LIN {X 0.002,Y -304.515,Z 1921.631,A 0.000,B 0.000,C 90.000,E1 293.567} C_DIS
LIN {X 0.065,Y -306.919,Z 1921.627,A 0.000,B 0.000,C 90.000,E1 292.898} C_DIS
LIN {X -0.021,Y -308.937,Z 1921.624,A 0.000,B 0.000,C 90.000,E1 292.259} C_DIS
LIN {X 0.067,Y -310.611,Z 1921.620,A 0.000,B 0.000,C 90.000,E1 291.589} C_DIS
LIN {X -0.119,Y -311.953,Z 1921.616,A 0.000,B 0.000,C 90.000,E1 290.972} C_DIS
LIN {X -0.004,Y -312.961,Z 1921.613,A 0.000,B 0.000,C 90.000,E1 290.301} C_DIS
LIN {X 0.121,Y -313.601,Z 1921.609,A 0.000,B 0.000,C 90.000,E1 289.631} C_DIS
LIN {X -0.147,Y -313.943,Z 1921.606,A 0.000,B 0.000,C 90.000,E1 289.033} C_DIS
LIN {X -0.011,Y -313.934,Z 1921.602,A 0.000,B 0.000,C 90.000,E1 288.362} C_DIS
LIN {X 0.123,Y -313.547,Z 1921.598,A 0.000,B 0.000,C 90.000,E1 287.692} C_DIS
LIN {X -0.136,Y -312.735,Z 1921.595,A 0.000,B 0.000,C 90.000,E1 287.094} C_DIS
LIN {X -0.097,Y -311.456,Z 1921.591,A 0.000,B 0.000,C 90.000,E1 286.441} C_DIS
LIN {X -0.092,Y -308.719,Z 1921.586,A 0.000,B 0.000,C 90.000,E1 285.536} C_DIS
LIN {X 0.054,Y -308.176,Z 1921.585,A 0.000,B 0.000,C 90.000,E1 285.371} C_DIS
LIN {X -0.002,Y -333.332,Z 1921.585,A 0.000,B 0.000,C 90.000,E1 285.371} C_DIS
LIN {X -0.184,Y -334.230,Z 1921.585,A 0.000,B 0.000,C 90.000,E1 285.371} C_DIS
LIN {X -0.037,Y -337.088,Z 1921.584,A 0.000,B 0.000,C 90.000,E1 285.134} C_DIS
LIN {X -0.135,Y -340.755,Z 1921.582,A 0.000,B 0.000,C 90.000,E1 284.717} C_DIS
LIN {X 0.172,Y -342.835,Z 1921.580,A 0.000,B 0.000,C 90.000,E1 284.356} C_DIS
LIN {X -0.028,Y -346.142,Z 1921.577,A 0.000,B 0.000,C 90.000,E1 283.772} C_DIS
LIN {X -0.039,Y -347.531,Z 1921.575,A 0.000,B 0.000,C 90.000,E1 283.467} C_DIS
LIN {X 0.137,Y -349.644,Z 1921.571,A 0.000,B 0.000,C 90.000,E1 282.827} C_DIS
LIN {X -0.010,Y -351.067,Z 1921.568,A 0.000,B 0.000,C 90.000,E1 282.243} C_DIS
LIN {X -0.151,Y -351.871,Z 1921.565,A 0.000,B 0.000,C 90.000,E1 281.658} C_DIS
LIN {X 0.132,Y -351.962,Z 1921.561,A 0.000,B 0.000,C 90.000,E1 281.007} C_DIS
LIN {X -0.062,Y -351.450,Z 1921.558,A 0.000,B 0.000,C 90.000,E1 280.433} C_DIS
LIN {X -0.187,Y -350.466,Z 1921.555,A 0.000,B 0.000,C 90.000,E1 279.849} C_DIS
LIN {X 0.028,Y -348.914,Z 1921.551,A 0.000,B 0.000,C 90.000,E1 279.208} C_DIS
LIN {X -0.110,Y -346.688,Z 1921.548,A 0.000,B 0.000,C 90.000,E1 278.624} C_DIS
LIN {X 0.028,Y -343.729,Z 1921.544,A 0.000,B 0.000,C 90.000,E1 277.992} C_DIS
LIN {X -0.057,Y -341.860,Z 1921.543,A 0.000,B 0.000,C 90.000,E1 277.701} C_DIS
LIN {X -0.142,Y -339.639,Z 1921.541,A 0.000,B 0.000,C 90.000,E1 277.409} C_DIS
LIN {X 0.056,Y -336.869,Z 1921.539,A 0.000,B 0.000,C 90.000,E1 277.068} C_DIS
LIN {X -0.039,Y -332.823,Z 1921.538,A 0.000,B 0.000,C 90.000,E1 276.777} C_DIS
LIN {X -0.008,Y -329.708,Z 1921.537,A 0.000,B 0.000,C 90.000,E1 276.663} C_DIS
LIN {X -0.039,Y -180.532,Z 1921.537,A 0.000,B 0.000,C 90.000,E1 276.663} C_DIS
LIN {X -0.091,Y -181.015,Z 1921.530,A 0.000,B 0.000,C 90.000,E1 275.511} C_DIS
LIN {X 0.078,Y -181.574,Z 1921.502,A 0.000,B 0.000,C 90.000,E1 270.401} C_DIS
LIN {X 0.054,Y -180.906,Z 1921.474,A 0.000,B 0.000,C 90.000,E1 265.355} C_DIS
LIN {X -0.052,Y -180.690,Z 1921.470,A 0.000,B 0.000,C 90.000,E1 264.546} C_DIS
LIN {X 0.026,Y -178.775,Z 1921.441,A 0.000,B 0.000,C 90.000,E1 259.454} C_DIS
LIN {X -0.071,Y -175.821,Z 1921.413,A 0.000,B 0.000,C 90.000,E1 254.393} C_DIS
LIN {X -0.071,Y -172.009,Z 1921.385,A 0.000,B 0.000,C 90.000,E1 249.263} C_DIS
LIN {X -0.094,Y -171.427,Z 1921.380,A 0.000,B 0.000,C 90.000,E1 248.411} C_DIS
LIN {X -0.038,Y -167.664,Z 1921.356,A 0.000,B 0.000,C 90.000,E1 244.076} C_DIS
LIN {X -0.098,Y -166.334,Z 1921.346,A 0.000,B 0.000,C 90.000,E1 242.359} C_DIS
LIN {X 0.035,Y -163.072,Z 1921.327,A 0.000,B 0.000,C 90.000,E1 238.820} C_DIS
LIN {X -0.054,Y -161.012,Z 1921.312,A 0.000,B 0.000,C 90.000,E1 236.215} C_DIS
LIN {X 0.056,Y -157.755,Z 1921.293,A 0.000,B 0.000,C 90.000,E1 232.637} C_DIS
LIN {X -0.005,Y -155.793,Z 1921.278,A 0.000,B 0.000,C 90.000,E1 229.989} C_DIS
LIN {X 0.050,Y -152.046,Z 1921.253,A 0.000,B 0.000,C 90.000,E1 225.486} C_DIS
LIN {X 0.067,Y -150.296,Z 1921.238,A 0.000,B 0.000,C 90.000,E1 222.771} C_DIS
LIN {X -0.008,Y -147.042,Z 1921.213,A 0.000,B 0.000,C 90.000,E1 218.257} C_DIS
LIN {X -0.016,Y -145.622,Z 1921.197,A 0.000,B 0.000,C 90.000,E1 215.518} C_DIS
LIN {X -0.016,Y -143.006,Z 1921.172,A 0.000,B 0.000,C 90.000,E1 210.924} C_DIS
LIN {X 0.041,Y -141.632,Z 1921.151,A 0.000,B 0.000,C 90.000,E1 207.206} C_DIS
LIN {X -0.034,Y -139.435,Z 1921.115,A 0.000,B 0.000,C 90.000,E1 200.737} C_DIS
LIN {X 0.020,Y -139.168,Z 1921.105,A 0.000,B 0.000,C 90.000,E1 198.852} C_DIS
LIN {X 0.053,Y -138.317,Z 1921.053,A 0.000,B 0.000,C 90.000,E1 189.500} C_DIS
LIN {X 0.065,Y -139.474,Z 1921.006,A 0.000,B 0.000,C 90.000,E1 181.088} C_DIS
LIN {X 0.006,Y -141.054,Z 1920.975,A 0.000,B 0.000,C 90.000,E1 175.527} C_DIS
LIN {X -0.040,Y -142.426,Z 1920.960,A 0.000,B 0.000,C 90.000,E1 172.761} C_DIS
LIN {X 0.021,Y -144.663,Z 1920.934,A 0.000,B 0.000,C 90.000,E1 168.117} C_DIS
LIN {X 0.005,Y -147.246,Z 1920.914,A 0.000,B 0.000,C 90.000,E1 164.448} C_DIS
LIN {X 0.022,Y -150.563,Z 1920.888,A 0.000,B 0.000,C 90.000,E1 159.880} C_DIS
LIN {X -0.038,Y -154.031,Z 1920.868,A 0.000,B 0.000,C 90.000,E1 156.282} C_DIS
LIN {X 0.030,Y -157.447,Z 1920.848,A 0.000,B 0.000,C 90.000,E1 152.666} C_DIS
LIN {X -0.021,Y -161.665,Z 1920.828,A 0.000,B 0.000,C 90.000,E1 149.125} C_DIS
LIN {X -0.004,Y -165.859,Z 1920.809,A 0.000,B 0.000,C 90.000,E1 145.595} C_DIS
LIN {X -0.012,Y -170.835,Z 1920.789,A 0.000,B 0.000,C 90.000,E1 142.110} C_DIS
LIN {X 0.035,Y -175.705,Z 1920.770,A 0.000,B 0.000,C 90.000,E1 138.647} C_DIS
LIN {X 0.026,Y -181.317,Z 1920.751,A 0.000,B 0.000,C 90.000,E1 135.243} C_DIS
LIN {X -0.102,Y -186.801,Z 1920.733,A 0.000,B 0.000,C 90.000,E1 131.919} C_DIS
LIN {X -0.033,Y -191.392,Z 1920.719,A 0.000,B 0.000,C 90.000,E1 129.402} C_DIS
LIN {X 0.050,Y -197.236,Z 1920.701,A 0.000,B 0.000,C 90.000,E1 126.091} C_DIS
LIN {X -0.027,Y -200.514,Z 1920.692,A 0.000,B 0.000,C 90.000,E1 124.485} C_DIS
LIN {X -0.010,Y -206.396,Z 1920.674,A 0.000,B 0.000,C 90.000,E1 121.258} C_DIS
LIN {X -0.024,Y -209.677,Z 1920.665,A 0.000,B 0.000,C 90.000,E1 119.667} C_DIS
LIN {X -0.003,Y -217.043,Z 1920.643,A 0.000,B 0.000,C 90.000,E1 115.720} C_DIS
LIN {X -0.050,Y -218.669,Z 1920.639,A 0.000,B 0.000,C 90.000,E1 114.951} C_DIS
LIN {X -0.129,Y -224.172,Z 1920.621,A 0.000,B 0.000,C 90.000,E1 111.844} C_DIS
LIN {X 0.065,Y -283.970,Z 1920.621,A 0.000,B 0.000,C 90.000,E1 111.791} C_DIS
LIN {X -0.075,Y -286.317,Z 1920.621,A 0.000,B 0.000,C 90.000,E1 111.770} C_DIS
LIN {X 0.024,Y -291.816,Z 1920.619,A 0.000,B 0.000,C 90.000,E1 111.408} C_DIS
LIN {X -0.148,Y -294.779,Z 1920.617,A 0.000,B 0.000,C 90.000,E1 111.099} C_DIS
LIN {X 0.031,Y -298.509,Z 1920.614,A 0.000,B 0.000,C 90.000,E1 110.429} C_DIS
LIN {X -0.011,Y -311.958,Z 1920.601,A 0.000,B 0.000,C 90.000,E1 108.127} C_DIS
LIN {X 0.151,Y -326.801,Z 1920.588,A 0.000,B 0.000,C 90.000,E1 105.843} C_DIS
LIN {X -0.150,Y -340.724,Z 1920.578,A 0.000,B 0.000,C 90.000,E1 104.008} C_DIS
LIN {X 0.141,Y -355.851,Z 1920.568,A 0.000,B 0.000,C 90.000,E1 102.119} C_DIS
LIN {X -0.028,Y -374.320,Z 1920.556,A 0.000,B 0.000,C 90.000,E1 100.141} C_DIS
LIN {X -0.206,Y -393.254,Z 1920.546,A 0.000,B 0.000,C 90.000,E1 98.341} C_DIS
LIN {X -0.087,Y -412.522,Z 1920.537,A 0.000,B 0.000,C 90.000,E1 96.663} C_DIS
LIN {X -0.058,Y -434.954,Z 1920.527,A 0.000,B 0.000,C 90.000,E1 94.935} C_DIS
LIN {X 0.159,Y -437.802,Z 1920.526,A 0.000,B 0.000,C 90.000,E1 94.702} C_DIS
LIN {X 0.165,Y -442.464,Z 1920.524,A 0.000,B 0.000,C 90.000,E1 94.302} C_DIS
LIN {X 0.194,Y -445.631,Z 1920.521,A 0.000,B 0.000,C 90.000,E1 93.841} C_DIS
LIN {X -0.076,Y -446.857,Z 1920.520,A 0.000,B 0.000,C 90.000,E1 93.612} C_DIS
LIN {X 0.103,Y -447.763,Z 1920.519,A 0.000,B 0.000,C 90.000,E1 93.326} C_DIS
LIN {X 0.063,Y -448.764,Z 1920.516,A 0.000,B 0.000,C 90.000,E1 92.808} C_DIS
LIN {X 0.007,Y -448.816,Z 1920.513,A 0.000,B 0.000,C 90.000,E1 92.293} C_DIS
LIN {X -0.027,Y -447.929,Z 1920.510,A 0.000,B 0.000,C 90.000,E1 91.776} C_DIS
LIN {X -0.077,Y -445.964,Z 1920.507,A 0.000,B 0.000,C 90.000,E1 91.260} C_DIS
LIN {X 0.057,Y -441.172,Z 1920.503,A 0.000,B 0.000,C 90.000,E1 90.458} C_DIS
LIN {X -0.085,Y -429.668,Z 1920.492,A 0.000,B 0.000,C 90.000,E1 88.625} C_DIS
LIN {X -0.011,Y -417.866,Z 1920.482,A 0.000,B 0.000,C 90.000,E1 86.731} C_DIS
LIN {X -0.167,Y -406.082,Z 1920.471,A 0.000,B 0.000,C 90.000,E1 84.837} C_DIS
LIN {X -0.095,Y -394.132,Z 1920.460,A 0.000,B 0.000,C 90.000,E1 82.875} C_DIS
LIN {X 0.170,Y -382.197,Z 1920.449,A 0.000,B 0.000,C 90.000,E1 80.849} C_DIS
LIN {X -0.136,Y -370.380,Z 1920.438,A 0.000,B 0.000,C 90.000,E1 78.870} C_DIS
LIN {X 0.056,Y -354.195,Z 1920.422,A 0.000,B 0.000,C 90.000,E1 75.880} C_DIS
LIN {X 0.111,Y -340.488,Z 1920.406,A 0.000,B 0.000,C 90.000,E1 73.142} C_DIS
LIN {X 0.021,Y -328.680,Z 1920.393,A 0.000,B 0.000,C 90.000,E1 70.678} C_DIS
LIN {X -0.086,Y -315.737,Z 1920.377,A 0.000,B 0.000,C 90.000,E1 67.847} C_DIS
LIN {X -0.010,Y -303.432,Z 1920.361,A 0.000,B 0.000,C 90.000,E1 64.921} C_DIS
LIN {X -0.036,Y -291.278,Z 1920.344,A 0.000,B 0.000,C 90.000,E1 61.948} C_DIS
LIN {X -0.011,Y -283.285,Z 1920.333,A 0.000,B 0.000,C 90.000,E1 59.921} C_DIS
LIN {X -0.002,Y -275.146,Z 1920.322,A 0.000,B 0.000,C 90.000,E1 57.867} C_DIS
LIN {X -0.012,Y -265.628,Z 1920.308,A 0.000,B 0.000,C 90.000,E1 55.435} C_DIS
LIN {X -0.032,Y -254.625,Z 1920.292,A 0.000,B 0.000,C 90.000,E1 52.603} C_DIS
LIN {X -0.032,Y -245.033,Z 1920.278,A 0.000,B 0.000,C 90.000,E1 50.070} C_DIS
LIN {X 0.006,Y -234.280,Z 1920.262,A 0.000,B 0.000,C 90.000,E1 47.106} C_DIS
LIN {X -0.080,Y -223.946,Z 1920.245,A 0.000,B 0.000,C 90.000,E1 44.109} C_DIS
LIN {X 0.065,Y -214.103,Z 1920.228,A 0.000,B 0.000,C 90.000,E1 40.987} C_DIS
LIN {X -0.014,Y -206.069,Z 1920.213,A 0.000,B 0.000,C 90.000,E1 38.257} C_DIS
LIN {X 0.108,Y -197.738,Z 1920.195,A 0.000,B 0.000,C 90.000,E1 35.025} C_DIS
LIN {X 0.015,Y -190.143,Z 1920.177,A 0.000,B 0.000,C 90.000,E1 31.799} C_DIS
LIN {X 0.025,Y -183.302,Z 1920.158,A 0.000,B 0.000,C 90.000,E1 28.487} C_DIS
LIN {X -0.061,Y -177.149,Z 1920.140,A 0.000,B 0.000,C 90.000,E1 25.155} C_DIS
LIN {X 0.038,Y -171.826,Z 1920.121,A 0.000,B 0.000,C 90.000,E1 21.716} C_DIS
LIN {X -0.028,Y -167.291,Z 1920.102,A 0.000,B 0.000,C 90.000,E1 18.290} C_DIS
LIN {X 0.066,Y -163.600,Z 1920.082,A 0.000,B 0.000,C 90.000,E1 14.773} C_DIS
LIN {X 0.088,Y -159.838,Z 1920.058,A 0.000,B 0.000,C 90.000,E1 10.366} C_DIS
LIN {X -0.012,Y -157.228,Z 1920.033,A 0.000,B 0.000,C 90.000,E1 5.967} C_DIS
LIN {X 0.000,Y -154.966,Z 1920.000,A 0.000,B 0.000,C 90.000,E1 360.000} C_DIS
LIN {X 0.054,Y -154.101,Z 1919.953,A 0.000,B 0.000,C 90.000,E1 351.432} C_DIS
LIN {X -0.028,Y -155.831,Z 1919.913,A 0.000,B 0.000,C 90.000,E1 344.283} C_DIS
LIN {X 0.034,Y -158.563,Z 1919.883,A 0.000,B 0.000,C 90.000,E1 338.901} C_DIS
LIN {X 0.048,Y -162.163,Z 1919.858,A 0.000,B 0.000,C 90.000,E1 334.460} C_DIS
LIN {X -0.045,Y -166.067,Z 1919.839,A 0.000,B 0.000,C 90.000,E1 330.973} C_DIS
LIN {X 0.052,Y -170.952,Z 1919.819,A 0.000,B 0.000,C 90.000,E1 327.454} C_DIS
LIN {X -0.036,Y -175.257,Z 1919.805,A 0.000,B 0.000,C 90.000,E1 324.895} C_DIS
LIN {X 0.018,Y -180.231,Z 1919.791,A 0.000,B 0.000,C 90.000,E1 322.316} C_DIS
LIN {X 0.017,Y -186.091,Z 1919.777,A 0.000,B 0.000,C 90.000,E1 319.784} C_DIS
LIN {X -0.017,Y -191.702,Z 1919.765,A 0.000,B 0.000,C 90.000,E1 317.715} C_DIS
LIN {X 0.020,Y -199.356,Z 1919.751,A 0.000,B 0.000,C 90.000,E1 315.243} C_DIS
LIN {X -0.077,Y -207.946,Z 1919.738,A 0.000,B 0.000,C 90.000,E1 312.852} C_DIS
LIN {X -0.098,Y -219.015,Z 1919.723,A 0.000,B 0.000,C 90.000,E1 310.092} C_DIS
LIN {X 0.025,Y -231.128,Z 1919.708,A 0.000,B 0.000,C 90.000,E1 307.363} C_DIS
LIN {X -0.157,Y -246.063,Z 1919.691,A 0.000,B 0.000,C 90.000,E1 304.405} C_DIS
LIN {X -0.153,Y -257.917,Z 1919.679,A 0.000,B 0.000,C 90.000,E1 302.212} C_DIS
LIN {X 0.088,Y -271.994,Z 1919.665,A 0.000,B 0.000,C 90.000,E1 299.667} C_DIS
LIN {X -0.138,Y -281.884,Z 1919.655,A 0.000,B 0.000,C 90.000,E1 297.975} C_DIS
LIN {X 0.035,Y -291.484,Z 1919.646,A 0.000,B 0.000,C 90.000,E1 296.232} C_DIS
LIN {X 0.116,Y -296.919,Z 1919.640,A 0.000,B 0.000,C 90.000,E1 295.207} C_DIS
LIN {X 0.118,Y -301.729,Z 1919.635,A 0.000,B 0.000,C 90.000,E1 294.207} C_DIS
LIN {X 0.004,Y -304.525,Z 1919.631,A 0.000,B 0.000,C 90.000,E1 293.567} C_DIS
LIN {X 0.065,Y -306.930,Z 1919.627,A 0.000,B 0.000,C 90.000,E1 292.898} C_DIS
LIN {X -0.020,Y -308.949,Z 1919.624,A 0.000,B 0.000,C 90.000,E1 292.259} C_DIS
LIN {X 0.069,Y -310.624,Z 1919.620,A 0.000,B 0.000,C 90.000,E1 291.589} C_DIS
LIN {X -0.117,Y -311.965,Z 1919.616,A 0.000,B 0.000,C 90.000,E1 290.972} C_DIS
LIN {X -0.002,Y -312.976,Z 1919.613,A 0.000,B 0.000,C 90.000,E1 290.301} C_DIS
LIN {X 0.122,Y -313.615,Z 1919.609,A 0.000,B 0.000,C 90.000,E1 289.631} C_DIS
LIN {X -0.146,Y -313.957,Z 1919.606,A 0.000,B 0.000,C 90.000,E1 289.033} C_DIS
LIN {X -0.010,Y -313.948,Z 1919.602,A 0.000,B 0.000,C 90.000,E1 288.362} C_DIS
LIN {X 0.027,Y -313.277,Z 1919.597,A 0.000,B 0.000,C 90.000,E1 287.457} C_DIS
LIN {X 0.090,Y -313.047,Z 1919.596,A 0.000,B 0.000,C 90.000,E1 287.275} C_DIS
LIN {X 0.056,Y -324.044,Z 1919.596,A 0.000,B 0.000,C 90.000,E1 287.275} C_DIS
LIN {X -0.132,Y -325.434,Z 1919.596,A 0.000,B 0.000,C 90.000,E1 287.275} C_DIS
LIN {X -0.141,Y -328.660,Z 1919.595,A 0.000,B 0.000,C 90.000,E1 287.094} C_DIS
LIN {X 0.053,Y -332.915,Z 1919.593,A 0.000,B 0.000,C 90.000,E1 286.677} C_DIS
LIN {X -0.176,Y -337.219,Z 1919.590,A 0.000,B 0.000,C 90.000,E1 286.205} C_DIS
LIN {X 0.007,Y -341.415,Z 1919.586,A 0.000,B 0.000,C 90.000,E1 285.552} C_DIS
LIN {X -0.110,Y -344.891,Z 1919.583,A 0.000,B 0.000,C 90.000,E1 284.954} C_DIS
LIN {X 0.129,Y -347.829,Z 1919.580,A 0.000,B 0.000,C 90.000,E1 284.300} C_DIS
LIN {X 0.049,Y -350.372,Z 1919.576,A 0.000,B 0.000,C 90.000,E1 283.703} C_DIS
LIN {X -0.099,Y -352.257,Z 1919.573,A 0.000,B 0.000,C 90.000,E1 283.119} C_DIS
LIN {X 0.107,Y -353.702,Z 1919.569,A 0.000,B 0.000,C 90.000,E1 282.479} C_DIS
LIN {X 0.056,Y -354.591,Z 1919.566,A 0.000,B 0.000,C 90.000,E1 281.883} C_DIS
LIN {X -0.062,Y -354.893,Z 1919.563,A 0.000,B 0.000,C 90.000,E1 281.299} C_DIS
LIN {X 0.172,Y -354.690,Z 1919.559,A 0.000,B 0.000,C 90.000,E1 280.658} C_DIS
LIN {X 0.061,Y -353.977,Z 1919.556,A 0.000,B 0.000,C 90.000,E1 280.074} C_DIS
LIN {X -0.112,Y -352.826,Z 1919.553,A 0.000,B 0.000,C 90.000,E1 279.500} C_DIS
LIN {X 0.119,Y -351.196,Z 1919.549,A 0.000,B 0.000,C 90.000,E1 278.859} C_DIS
LIN {X -0.007,Y -349.066,Z 1919.546,A 0.000,B 0.000,C 90.000,E1 278.276} C_DIS
LIN {X 0.152,Y -346.346,Z 1919.543,A 0.000,B 0.000,C 90.000,E1 277.644} C_DIS
LIN {X -0.050,Y -342.831,Z 1919.539,A 0.000,B 0.000,C 90.000,E1 277.068} C_DIS
LIN {X -0.138,Y -340.766,Z 1919.537,A 0.000,B 0.000,C 90.000,E1 276.777} C_DIS
LIN {X 0.111,Y -338.329,Z 1919.536,A 0.000,B 0.000,C 90.000,E1 276.429} C_DIS
LIN {X -0.027,Y -335.363,Z 1919.534,A 0.000,B 0.000,C 90.000,E1 276.144} C_DIS
LIN {X -0.128,Y -331.749,Z 1919.532,A 0.000,B 0.000,C 90.000,E1 275.853} C_DIS
LIN {X 0.107,Y -328.073,Z 1919.531,A 0.000,B 0.000,C 90.000,E1 275.568} C_DIS
LIN {X 0.045,Y -321.865,Z 1919.530,A 0.000,B 0.000,C 90.000,E1 275.334} C_DIS
LIN {X -0.049,Y -320.654,Z 1919.530,A 0.000,B 0.000,C 90.000,E1 275.334} C_DIS
LIN {X -0.054,Y -181.040,Z 1919.530,A 0.000,B 0.000,C 90.000,E1 275.334} C_DIS
LIN {X -0.051,Y -181.567,Z 1919.500,A 0.000,B 0.000,C 90.000,E1 270.057} C_DIS
LIN {X -0.063,Y -180.860,Z 1919.472,A 0.000,B 0.000,C 90.000,E1 265.008} C_DIS
LIN {X -0.010,Y -178.971,Z 1919.444,A 0.000,B 0.000,C 90.000,E1 259.926} C_DIS
LIN {X 0.001,Y -177.930,Z 1919.435,A 0.000,B 0.000,C 90.000,E1 258.229} C_DIS
LIN {X 0.016,Y -175.568,Z 1919.411,A 0.000,B 0.000,C 90.000,E1 253.976} C_DIS
LIN {X 0.023,Y -172.297,Z 1919.387,A 0.000,B 0.000,C 90.000,E1 249.699} C_DIS
LIN {X 0.000,Y -171.776,Z 1919.382,A 0.000,B 0.000,C 90.000,E1 248.847} C_DIS
LIN {X -0.027,Y -168.705,Z 1919.363,A 0.000,B 0.000,C 90.000,E1 245.409} C_DIS
LIN {X 0.011,Y -166.769,Z 1919.349,A 0.000,B 0.000,C 90.000,E1 242.794} C_DIS
LIN {X 0.070,Y -162.748,Z 1919.325,A 0.000,B 0.000,C 90.000,E1 238.408} C_DIS
LIN {X -0.092,Y -161.439,Z 1919.315,A 0.000,B 0.000,C 90.000,E1 236.707} C_DIS
LIN {X -0.050,Y -157.432,Z 1919.290,A 0.000,B 0.000,C 90.000,E1 232.271} C_DIS
LIN {X -0.015,Y -155.438,Z 1919.275,A 0.000,B 0.000,C 90.000,E1 229.585} C_DIS
LIN {X 0.034,Y -151.759,Z 1919.250,A 0.000,B 0.000,C 90.000,E1 225.081} C_DIS
LIN {X 0.045,Y -149.960,Z 1919.235,A 0.000,B 0.000,C 90.000,E1 222.366} C_DIS
LIN {X 0.072,Y -146.801,Z 1919.210,A 0.000,B 0.000,C 90.000,E1 217.810} C_DIS
LIN {X -0.028,Y -145.376,Z 1919.195,A 0.000,B 0.000,C 90.000,E1 215.105} C_DIS
LIN {X -0.035,Y -142.439,Z 1919.164,A 0.000,B 0.000,C 90.000,E1 209.589} C_DIS
LIN {X 0.011,Y -141.430,Z 1919.149,A 0.000,B 0.000,C 90.000,E1 206.796} C_DIS
LIN {X -0.007,Y -139.365,Z 1919.113,A 0.000,B 0.000,C 90.000,E1 200.301} C_DIS
LIN {X -0.021,Y -138.810,Z 1919.097,A 0.000,B 0.000,C 90.000,E1 197.511} C_DIS
LIN {X 0.029,Y -138.351,Z 1919.056,A 0.000,B 0.000,C 90.000,E1 190.018} C_DIS
LIN {X 0.006,Y -139.541,Z 1919.004,A 0.000,B 0.000,C 90.000,E1 180.688} C_DIS
LIN {X -0.042,Y -141.237,Z 1918.973,A 0.000,B 0.000,C 90.000,E1 175.122} C_DIS
LIN {X 0.058,Y -142.608,Z 1918.957,A 0.000,B 0.000,C 90.000,E1 172.299} C_DIS
LIN {X 0.011,Y -144.920,Z 1918.932,A 0.000,B 0.000,C 90.000,E1 167.701} C_DIS
LIN {X 0.003,Y -147.548,Z 1918.911,A 0.000,B 0.000,C 90.000,E1 164.031} C_DIS
LIN {X 0.035,Y -150.151,Z 1918.891,A 0.000,B 0.000,C 90.000,E1 160.369} C_DIS
LIN {X 0.045,Y -153.521,Z 1918.871,A 0.000,B 0.000,C 90.000,E1 156.741} C_DIS
LIN {X -0.034,Y -157.886,Z 1918.846,A 0.000,B 0.000,C 90.000,E1 152.281} C_DIS
LIN {X -0.080,Y -162.173,Z 1918.826,A 0.000,B 0.000,C 90.000,E1 148.742} C_DIS
LIN {X 0.035,Y -166.382,Z 1918.807,A 0.000,B 0.000,C 90.000,E1 145.182} C_DIS
LIN {X 0.036,Y -171.398,Z 1918.787,A 0.000,B 0.000,C 90.000,E1 141.698} C_DIS
LIN {X 0.076,Y -176.311,Z 1918.768,A 0.000,B 0.000,C 90.000,E1 138.243} C_DIS
LIN {X -0.055,Y -180.598,Z 1918.754,A 0.000,B 0.000,C 90.000,E1 135.729} C_DIS
LIN {X -0.077,Y -186.000,Z 1918.735,A 0.000,B 0.000,C 90.000,E1 132.366} C_DIS
LIN {X -0.022,Y -190.635,Z 1918.721,A 0.000,B 0.000,C 90.000,E1 129.850} C_DIS
LIN {X -0.116,Y -196.386,Z 1918.703,A 0.000,B 0.000,C 90.000,E1 126.583} C_DIS
LIN {X -0.040,Y -201.176,Z 1918.689,A 0.000,B 0.000,C 90.000,E1 124.119} C_DIS
LIN {X 0.056,Y -207.123,Z 1918.672,A 0.000,B 0.000,C 90.000,E1 120.875} C_DIS
LIN {X 0.056,Y -210.399,Z 1918.663,A 0.000,B 0.000,C 90.000,E1 119.283} C_DIS
LIN {X -0.041,Y -216.186,Z 1918.645,A 0.000,B 0.000,C 90.000,E1 116.155} C_DIS
LIN {X -0.032,Y -219.350,Z 1918.637,A 0.000,B 0.000,C 90.000,E1 114.591} C_DIS
LIN {X -0.103,Y -224.160,Z 1918.621,A 0.000,B 0.000,C 90.000,E1 111.844} C_DIS
LIN {X 0.081,Y -283.777,Z 1918.621,A 0.000,B 0.000,C 90.000,E1 111.791} C_DIS
LIN {X 0.082,Y -285.206,Z 1918.621,A 0.000,B 0.000,C 90.000,E1 111.770} C_DIS
LIN {X 0.032,Y -290.971,Z 1918.619,A 0.000,B 0.000,C 90.000,E1 111.482} C_DIS
LIN {X 0.081,Y -294.043,Z 1918.618,A 0.000,B 0.000,C 90.000,E1 111.153} C_DIS
LIN {X -0.153,Y -297.714,Z 1918.614,A 0.000,B 0.000,C 90.000,E1 110.610} C_DIS
LIN {X 0.157,Y -311.095,Z 1918.601,A 0.000,B 0.000,C 90.000,E1 108.236} C_DIS
LIN {X -0.104,Y -325.850,Z 1918.589,A 0.000,B 0.000,C 90.000,E1 106.024} C_DIS
LIN {X -0.019,Y -339.690,Z 1918.578,A 0.000,B 0.000,C 90.000,E1 104.120} C_DIS
LIN {X -0.170,Y -354.728,Z 1918.568,A 0.000,B 0.000,C 90.000,E1 102.299} C_DIS
LIN {X 0.006,Y -373.168,Z 1918.557,A 0.000,B 0.000,C 90.000,E1 100.254} C_DIS
LIN {X 0.141,Y -392.077,Z 1918.547,A 0.000,B 0.000,C 90.000,E1 98.398} C_DIS
LIN {X -0.203,Y -411.326,Z 1918.537,A 0.000,B 0.000,C 90.000,E1 96.777} C_DIS
LIN {X 0.179,Y -433.736,Z 1918.528,A 0.000,B 0.000,C 90.000,E1 94.992} C_DIS
LIN {X 0.166,Y -439.382,Z 1918.526,A 0.000,B 0.000,C 90.000,E1 94.588} C_DIS
LIN {X -0.059,Y -441.665,Z 1918.525,A 0.000,B 0.000,C 90.000,E1 94.416} C_DIS
LIN {X -0.098,Y -445.192,Z 1918.522,A 0.000,B 0.000,C 90.000,E1 93.955} C_DIS
LIN {X 0.076,Y -446.525,Z 1918.520,A 0.000,B 0.000,C 90.000,E1 93.669} C_DIS
LIN {X -0.195,Y -447.519,Z 1918.519,A 0.000,B 0.000,C 90.000,E1 93.440} C_DIS
LIN {X 0.211,Y -448.666,Z 1918.516,A 0.000,B 0.000,C 90.000,E1 92.865} C_DIS
LIN {X 0.152,Y -448.851,Z 1918.513,A 0.000,B 0.000,C 90.000,E1 92.350} C_DIS
LIN {X 0.104,Y -448.103,Z 1918.510,A 0.000,B 0.000,C 90.000,E1 91.835} C_DIS
LIN {X 0.069,Y -446.312,Z 1918.507,A 0.000,B 0.000,C 90.000,E1 91.318} C_DIS
LIN {X -0.180,Y -444.923,Z 1918.506,A 0.000,B 0.000,C 90.000,E1 91.088} C_DIS
LIN {X 0.191,Y -433.427,Z 1918.496,A 0.000,B 0.000,C 90.000,E1 89.198} C_DIS
LIN {X 0.199,Y -423.392,Z 1918.487,A 0.000,B 0.000,C 90.000,E1 87.593} C_DIS
LIN {X 0.142,Y -411.614,Z 1918.476,A 0.000,B 0.000,C 90.000,E1 85.698} C_DIS
LIN {X -0.201,Y -401.450,Z 1918.467,A 0.000,B 0.000,C 90.000,E1 84.090} C_DIS
LIN {X 0.163,Y -389.472,Z 1918.456,A 0.000,B 0.000,C 90.000,E1 82.072} C_DIS
LIN {X -0.006,Y -377.587,Z 1918.445,A 0.000,B 0.000,C 90.000,E1 80.095} C_DIS
LIN {X -0.028,Y -360.994,Z 1918.429,A 0.000,B 0.000,C 90.000,E1 77.173} C_DIS
LIN {X 0.046,Y -345.419,Z 1918.412,A 0.000,B 0.000,C 90.000,E1 74.157} C_DIS
LIN {X 0.081,Y -333.484,Z 1918.398,A 0.000,B 0.000,C 90.000,E1 71.692} C_DIS
LIN {X -0.022,Y -323.249,Z 1918.386,A 0.000,B 0.000,C 90.000,E1 69.518} C_DIS
LIN {X 0.052,Y -309.206,Z 1918.368,A 0.000,B 0.000,C 90.000,E1 66.305} C_DIS
